gfCNCPoint3[22820] = {X 293.7166, Y 53.8663, Z -4.6667, A 0.000, B 0.000, C 0.000 }
gfCNCPoint3[22821] = {X 294.6128, Y 54.1799, Z -4.6667, A 0.000, B 0.000, C 0.000 }
gfCNCPoint3[22822] = {X 295.4167, Y 54.6850, Z -4.6667, A 0.000, B 0.000, C 0.000 }
gfCNCPoint3[22823] = {X 296.0881, Y 55.3564, Z -4.6667, A 0.000, B 0.000, C 0.000 }
gfCNCPoint3[22824] = {X 296.5932, Y 56.1603, Z -4.6667, A 0.000, B 0.000, C 0.000 }
gfCNCPoint3[22825] = {X 296.9068, Y 57.0565, Z -4.6667, A 0.000, B 0.000, C 0.000 }
gfCNCPoint3[22826] = {X 297.0131, Y 58.0000, Z -4.6667, A 0.000, B 0.000, C 0.000 }
gfCNCPoint3[22827] = {X 297.0131, Y 58.9348, Z -4.6667, A 0.000, B 0.000, C 0.000 }
gfCNCPoint3[22828] = {X 296.9205, Y 59.8045, Z -4.6667, A 0.000, B 0.000, C 0.000 }
gfCNCPoint3[22829] = {X 296.6522, Y 60.6370, Z -4.6667, A 0.000, B 0.000, C 0.000 }
gfCNCPoint3[22830] = {X 296.2193, Y 61.3970, Z -4.6667, A 0.000, B 0.000, C 0.000 }
gfCNCPoint3[22831] = {X 295.6403, Y 62.0524, Z -4.6667, A 0.000, B 0.000, C 0.000 }
gfCNCPoint3[22832] = {X 294.9395, Y 62.5757, Z -4.6667, A 0.000, B 0.000, C 0.000 }
gfCNCPoint3[22833] = {X 294.1465, Y 62.9448, Z -4.6667, A 0.000, B 0.000, C 0.000 }
gfCNCPoint3[22834] = {X 293.2949, Y 63.1439, Z -4.6667, A 0.000, B 0.000, C 0.000 }
gfCNCPoint3[22835] = {X 293.3045, Y 92.8506, Z -4.6667, A 0.000, B 0.000, C 0.000 }
gfCNCPoint3[22836] = {X 294.1540, Y 93.0538, Z -4.6667, A 0.000, B 0.000, C 0.000 }
gfCNCPoint3[22837] = {X 294.9444, Y 93.4255, Z -4.6667, A 0.000, B 0.000, C 0.000 }
gfCNCPoint3[22838] = {X 295.6427, Y 93.9502, Z -4.6667, A 0.000, B 0.000, C 0.000 }
gfCNCPoint3[22839] = {X 296.2197, Y 94.6059, Z -4.6667, A 0.000, B 0.000, C 0.000 }
gfCNCPoint3[22840] = {X 296.6513, Y 95.3652, Z -4.6667, A 0.000, B 0.000, C 0.000 }
gfCNCPoint3[22841] = {X 296.9195, Y 96.1965, Z -4.6667, A 0.000, B 0.000, C 0.000 }
gfCNCPoint3[22842] = {X 297.0131, Y 97.0649, Z -4.6667, A 0.000, B 0.000, C 0.000 }
gfCNCPoint3[22843] = {X 297.0131, Y 98.0000, Z -4.6667, A 0.000, B 0.000, C 0.000 }
gfCNCPoint3[22844] = {X 296.9068, Y 98.9435, Z -4.6667, A 0.000, B 0.000, C 0.000 }
gfCNCPoint3[22845] = {X 296.5932, Y 99.8397, Z -4.6667, A 0.000, B 0.000, C 0.000 }
gfCNCPoint3[22846] = {X 296.0881, Y 100.6436, Z -4.6667, A 0.000, B 0.000, C 0.000 }
gfCNCPoint3[22847] = {X 295.4167, Y 101.3150, Z -4.6667, A 0.000, B 0.000, C 0.000 }
gfCNCPoint3[22848] = {X 294.6128, Y 101.8201, Z -4.6667, A 0.000, B 0.000, C 0.000 }
gfCNCPoint3[22849] = {X 293.7166, Y 102.1337, Z -4.6667, A 0.000, B 0.000, C 0.000 }
gfCNCPoint3[22850] = {X 292.7731, Y 102.2400, Z -4.6667, A 0.000, B 0.000, C 0.000 }
gfCNCPoint3[22851] = {X 276.2327, Y 102.2400, Z -4.6667, A 0.000, B 0.000, C 0.000 }
gfCNCPoint3[22852] = {X 275.2892, Y 102.1337, Z -4.6667, A 0.000, B 0.000, C 0.000 }
gfCNCPoint3[22853] = {X 274.3930, Y 101.8201, Z -4.6667, A 0.000, B 0.000, C 0.000 }
gfCNCPoint3[22854] = {X 273.5891, Y 101.3150, Z -4.6667, A 0.000, B 0.000, C 0.000 }
gfCNCPoint3[22855] = {X 272.9177, Y 100.6436, Z -4.6667, A 0.000, B 0.000, C 0.000 }
gfCNCPoint3[22856] = {X 272.4126, Y 99.8397, Z -4.6667, A 0.000, B 0.000, C 0.000 }
gfCNCPoint3[22857] = {X 272.0990, Y 98.9435, Z -4.6667, A 0.000, B 0.000, C 0.000 }
gfCNCPoint3[22858] = {X 271.9927, Y 98.0000, Z -4.6667, A 0.000, B 0.000, C 0.000 }
gfCNCPoint3[22859] = {X 271.9927, Y 97.0659, Z -4.6667, A 0.000, B 0.000, C 0.000 }
gfCNCPoint3[22860] = {X 272.0830, Y 96.1956, Z -4.6667, A 0.000, B 0.000, C 0.000 }
gfCNCPoint3[22861] = {X 272.3500, Y 95.3624, Z -4.6667, A 0.000, B 0.000, C 0.000 }
gfCNCPoint3[22862] = {X 272.7823, Y 94.6017, Z -4.6667, A 0.000, B 0.000, C 0.000 }
gfCNCPoint3[22863] = {X 273.3615, Y 93.9460, Z -4.6667, A 0.000, B 0.000, C 0.000 }
gfCNCPoint3[22864] = {X 274.0630, Y 93.4231, Z -4.6667, A 0.000, B 0.000, C 0.000 }
gfCNCPoint3[22865] = {X 274.8569, Y 93.0553, Z -4.6667, A 0.000, B 0.000, C 0.000 }
gfCNCPoint3[22866] = {X 275.7094, Y 92.8584, Z -4.6667, A 0.000, B 0.000, C 0.000 }
gfCNCPoint3[22867] = {X 275.7094, Y 85.5404, Z -4.6667, A 0.000, B 0.000, C 0.000 }
gfCNCPoint3[22868] = {X 262.6312, Y 80.4137, Z -4.6667, A 0.000, B 0.000, C 0.000 }
gfCNCPoint3[22869] = {X 262.2340, Y 80.6642, Z -4.6667, A 0.000, B 0.000, C 0.000 }
gfCNCPoint3[22870] = {X 237.7164, Y 96.5448, Z -4.6667, A 0.000, B 0.000, C 0.000 }
gfCNCPoint3[22871] = {X 237.7198, Y 97.0651, Z -4.6667, A 0.000, B 0.000, C 0.000 }
gfCNCPoint3[22872] = {X 237.7198, Y 98.0000, Z -4.6667, A 0.000, B 0.000, C 0.000 }
gfCNCPoint3[22873] = {X 237.6135, Y 98.9435, Z -4.6667, A 0.000, B 0.000, C 0.000 }
gfCNCPoint3[22874] = {X 237.2999, Y 99.8397, Z -4.6667, A 0.000, B 0.000, C 0.000 }
gfCNCPoint3[22875] = {X 236.7948, Y 100.6436, Z -4.6667, A 0.000, B 0.000, C 0.000 }
gfCNCPoint3[22876] = {X 236.1234, Y 101.3150, Z -4.6667, A 0.000, B 0.000, C 0.000 }
gfCNCPoint3[22877] = {X 235.3195, Y 101.8201, Z -4.6667, A 0.000, B 0.000, C 0.000 }
gfCNCPoint3[22878] = {X 234.4233, Y 102.1337, Z -4.6667, A 0.000, B 0.000, C 0.000 }
gfCNCPoint3[22879] = {X 233.4798, Y 102.2400, Z -4.6667, A 0.000, B 0.000, C 0.000 }
gfCNCPoint3[22880] = {X 214.1790, Y 102.2400, Z -4.6667, A 0.000, B 0.000, C 0.000 }
gfCNCPoint3[22881] = {X 213.7861, Y 102.2218, Z -4.6667, A 0.000, B 0.000, C 0.000 }
gfCNCPoint3[22882] = {X 213.3966, Y 102.1672, Z -4.6667, A 0.000, B 0.000, C 0.000 }
gfCNCPoint3[22883] = {X 213.0070, Y 102.2218, Z -4.6667, A 0.000, B 0.000, C 0.000 }
gfCNCPoint3[22884] = {X 212.6141, Y 102.2400, Z -4.6667, A 0.000, B 0.000, C 0.000 }
gfCNCPoint3[22885] = {X 194.9870, Y 102.2400, Z -4.6667, A 0.000, B 0.000, C 0.000 }
gfCNCPoint3[22886] = {X 194.0435, Y 102.1337, Z -4.6667, A 0.000, B 0.000, C 0.000 }
gfCNCPoint3[22887] = {X 193.1473, Y 101.8201, Z -4.6667, A 0.000, B 0.000, C 0.000 }
gfCNCPoint3[22888] = {X 192.3434, Y 101.3150, Z -4.6667, A 0.000, B 0.000, C 0.000 }
gfCNCPoint3[22889] = {X 191.6720, Y 100.6436, Z -4.6667, A 0.000, B 0.000, C 0.000 }
gfCNCPoint3[22890] = {X 191.1669, Y 99.8397, Z -4.6667, A 0.000, B 0.000, C 0.000 }
gfCNCPoint3[22891] = {X 190.8533, Y 98.9435, Z -4.6667, A 0.000, B 0.000, C 0.000 }
gfCNCPoint3[22892] = {X 190.7470, Y 98.0000, Z -4.6667, A 0.000, B 0.000, C 0.000 }
gfCNCPoint3[22893] = {X 190.7470, Y 97.0659, Z -4.6667, A 0.000, B 0.000, C 0.000 }
gfCNCPoint3[22894] = {X 190.8557, Y 96.1118, Z -4.6667, A 0.000, B 0.000, C 0.000 }
gfCNCPoint3[22895] = {X 191.1764, Y 95.2065, Z -4.6667, A 0.000, B 0.000, C 0.000 }
gfCNCPoint3[22896] = {X 191.6926, Y 94.3967, Z -4.6667, A 0.000, B 0.000, C 0.000 }
gfCNCPoint3[22897] = {X 188.5999, Y 91.0202, Z -4.6667, A 0.000, B 0.000, C 0.000 }
gfCNCPoint3[22898] = {X 150.0543, Y 91.0202, Z -4.6667, A 0.000, B 0.000, C 0.000 }
gfCNCPoint3[22899] = {X 147.0396, Y 94.3601, Z -4.6667, A 0.000, B 0.000, C 0.000 }
gfCNCPoint3[22900] = {X 147.5718, Y 95.1783, Z -4.6667, A 0.000, B 0.000, C 0.000 }
gfCNCPoint3[22901] = {X 147.9041, Y 96.0960, Z -4.6667, A 0.000, B 0.000, C 0.000 }
gfCNCPoint3[22902] = {X 148.0191, Y 97.0652, Z -4.6667, A 0.000, B 0.000, C 0.000 }
gfCNCPoint3[22903] = {X 148.0191, Y 98.0000, Z -4.6667, A 0.000, B 0.000, C 0.000 }
gfCNCPoint3[22904] = {X 147.9128, Y 98.9435, Z -4.6667, A 0.000, B 0.000, C 0.000 }
gfCNCPoint3[22905] = {X 147.5992, Y 99.8397, Z -4.6667, A 0.000, B 0.000, C 0.000 }
gfCNCPoint3[22906] = {X 147.0941, Y 100.6436, Z -4.6667, A 0.000, B 0.000, C 0.000 }
gfCNCPoint3[22907] = {X 146.4227, Y 101.3150, Z -4.6667, A 0.000, B 0.000, C 0.000 }
gfCNCPoint3[22908] = {X 145.6188, Y 101.8201, Z -4.6667, A 0.000, B 0.000, C 0.000 }
gfCNCPoint3[22909] = {X 144.7226, Y 102.1337, Z -4.6667, A 0.000, B 0.000, C 0.000 }
gfCNCPoint3[22910] = {X 143.7791, Y 102.2400, Z -4.6667, A 0.000, B 0.000, C 0.000 }
gfCNCPoint3[22911] = {X 125.0000, Y 102.2400, Z -4.6667, A 0.000, B 0.000, C 0.000 }
gfCNCPoint3[22912] = {X 124.0565, Y 102.1337, Z -4.6667, A 0.000, B 0.000, C 0.000 }
gfCNCPoint3[22913] = {X 123.1603, Y 101.8201, Z -4.6667, A 0.000, B 0.000, C 0.000 }
gfCNCPoint3[22914] = {X 122.3564, Y 101.3150, Z -4.6667, A 0.000, B 0.000, C 0.000 }
gfCNCPoint3[22915] = {X 121.6850, Y 100.6436, Z -4.6667, A 0.000, B 0.000, C 0.000 }
gfCNCPoint3[22916] = {X 121.1799, Y 99.8397, Z -4.6667, A 0.000, B 0.000, C 0.000 }
gfCNCPoint3[22917] = {X 120.8663, Y 98.9435, Z -4.6667, A 0.000, B 0.000, C 0.000 }
gfCNCPoint3[22918] = {X 120.7600, Y 98.0000, Z -4.6667, A 0.000, B 0.000, C 0.000 }
gfCNCPoint3[22919] = {X 120.7600, Y 97.0659, Z -4.6667, A 0.000, B 0.000, C 0.000 }
gfCNCPoint3[22920] = {X 120.8618, Y 96.1422, Z -4.6667, A 0.000, B 0.000, C 0.000 }
gfCNCPoint3[22921] = {X 121.1625, Y 95.2629, Z -4.6667, A 0.000, B 0.000, C 0.000 }
gfCNCPoint3[22922] = {X 121.6474, Y 94.4702, Z -4.6667, A 0.000, B 0.000, C 0.000 }
gfCNCPoint3[22923] = {X 122.2934, Y 93.8022, Z -4.6667, A 0.000, B 0.000, C 0.000 }
gfCNCPoint3[22924] = {X 123.0694, Y 93.2910, Z -4.6667, A 0.000, B 0.000, C 0.000 }
gfCNCPoint3[22925] = {X 123.9382, Y 92.9610, Z -4.6667, A 0.000, B 0.000, C 0.000 }
gfCNCPoint3[22926] = {X 124.8579, Y 92.8283, Z -4.6667, A 0.000, B 0.000, C 0.000 }
gfCNCPoint3[22927] = {X 124.8975, Y 92.8108, Z -4.6667, A 0.000, B 0.000, C 0.000 }
gfCNCPoint3[22928] = {X 124.9396, Y 92.8006, Z -4.6667, A 0.000, B 0.000, C 0.000 }
gfCNCPoint3[22929] = {X 125.4606, Y 92.7233, Z -4.6667, A 0.000, B 0.000, C 0.000 }
gfCNCPoint3[22930] = {X 126.3060, Y 92.5807, Z -4.6667, A 0.000, B 0.000, C 0.000 }
gfCNCPoint3[22931] = {X 127.1395, Y 92.3799, Z -4.6667, A 0.000, B 0.000, C 0.000 }
gfCNCPoint3[22932] = {X 128.3715, Y 91.2197, Z -4.6667, A 0.000, B 0.000, C 0.000 }
gfCNCPoint3[22933] = {X 129.5383, Y 89.9938, Z -4.6667, A 0.000, B 0.000, C 0.000 }
gfCNCPoint3[22934] = {X 140.7393, Y 77.6936, Z -4.6667, A 0.000, B 0.000, C 0.000 }
gfCNCPoint3[22935] = {X 137.7818, Y 75.0004, Z -4.6667, A 0.000, B 0.000, C 0.000 }
gfCNCPoint3[22936] = {X 140.7985, Y 77.7475, Z -4.6667, A 0.000, B 0.000, C 0.000 }
gfCNCPoint3[22937] = {X 155.8335, Y 61.2369, Z -4.6667, A 0.000, B 0.000, C 0.000 }
gfCNCPoint3[22938] = {X 155.4565, Y 60.5305, Z -4.6667, A 0.000, B 0.000, C 0.000 }
gfCNCPoint3[22939] = {X 155.2218, Y 59.7648, Z -4.6667, A 0.000, B 0.000, C 0.000 }
gfCNCPoint3[22940] = {X 155.1381, Y 58.9684, Z -4.6667, A 0.000, B 0.000, C 0.000 }
gfCNCPoint3[22941] = {X 155.1380, Y 58.0000, Z -4.6667, A 0.000, B 0.000, C 0.000 }
gfCNCPoint3[22942] = {X 155.2423, Y 57.0743, Z -4.6667, A 0.000, B 0.000, C 0.000 }
gfCNCPoint3[22943] = {X 155.5499, Y 56.1950, Z -4.6667, A 0.000, B 0.000, C 0.000 }
gfCNCPoint3[22944] = {X 156.0455, Y 55.4063, Z -4.6667, A 0.000, B 0.000, C 0.000 }
gfCNCPoint3[22945] = {X 156.7042, Y 54.7476, Z -4.6667, A 0.000, B 0.000, C 0.000 }
gfCNCPoint3[22946] = {X 157.4930, Y 54.2520, Z -4.6667, A 0.000, B 0.000, C 0.000 }
gfCNCPoint3[22947] = {X 158.3723, Y 53.9443, Z -4.6667, A 0.000, B 0.000, C 0.000 }
gfCNCPoint3[22948] = {X 159.2980, Y 53.8400, Z -4.6667, A 0.000, B 0.000, C 0.000 }
gfCNCPoint3[22949] = {X 178.5335, Y 53.8400, Z -4.6667, A 0.000, B 0.000, C 0.000 }
gfCNCPoint3[22950] = {X 179.4592, Y 53.9443, Z -4.6667, A 0.000, B 0.000, C 0.000 }
gfCNCPoint3[22951] = {X 180.3385, Y 54.2520, Z -4.6667, A 0.000, B 0.000, C 0.000 }
gfCNCPoint3[22952] = {X 181.1272, Y 54.7476, Z -4.6667, A 0.000, B 0.000, C 0.000 }
gfCNCPoint3[22953] = {X 181.7859, Y 55.4063, Z -4.6667, A 0.000, B 0.000, C 0.000 }
gfCNCPoint3[22954] = {X 182.2815, Y 56.1950, Z -4.6667, A 0.000, B 0.000, C 0.000 }
gfCNCPoint3[22955] = {X 182.5892, Y 57.0743, Z -4.6667, A 0.000, B 0.000, C 0.000 }
gfCNCPoint3[22956] = {X 182.6935, Y 58.0000, Z -4.6667, A 0.000, B 0.000, C 0.000 }
gfCNCPoint3[22957] = {X 182.6935, Y 58.9342, Z -4.6667, A 0.000, B 0.000, C 0.000 }
gfCNCPoint3[22958] = {X 182.6160, Y 59.7334, Z -4.6667, A 0.000, B 0.000, C 0.000 }
gfCNCPoint3[22959] = {X 182.3864, Y 60.5029, Z -4.6667, A 0.000, B 0.000, C 0.000 }
gfCNCPoint3[22960] = {X 182.0132, Y 61.2138, Z -4.6667, A 0.000, B 0.000, C 0.000 }
gfCNCPoint3[22961] = {X 209.3608, Y 91.0622, Z -4.6667, A 0.000, B 0.000, C 0.000 }
gfCNCPoint3[22962] = {X 210.0261, Y 91.7373, Z -4.6667, A 0.000, B 0.000, C 0.000 }
gfCNCPoint3[22963] = {X 210.7388, Y 92.3620, Z -4.6667, A 0.000, B 0.000, C 0.000 }
gfCNCPoint3[22964] = {X 211.0469, Y 92.5567, Z -4.6667, A 0.000, B 0.000, C 0.000 }
gfCNCPoint3[22965] = {X 211.3924, Y 92.6727, Z -4.6667, A 0.000, B 0.000, C 0.000 }
gfCNCPoint3[22966] = {X 213.3994, Y 92.9858, Z -4.6667, A 0.000, B 0.000, C 0.000 }
gfCNCPoint3[22967] = {X 214.4547, Y 92.8962, Z -4.6667, A 0.000, B 0.000, C 0.000 }
gfCNCPoint3[22968] = {X 215.5121, Y 92.8355, Z -4.6667, A 0.000, B 0.000, C 0.000 }
gfCNCPoint3[22969] = {X 216.2108, Y 92.7589, Z -4.6667, A 0.000, B 0.000, C 0.000 }
gfCNCPoint3[22970] = {X 216.8837, Y 92.5552, Z -4.6667, A 0.000, B 0.000, C 0.000 }
gfCNCPoint3[22971] = {X 217.5077, Y 92.2315, Z -4.6667, A 0.000, B 0.000, C 0.000 }
gfCNCPoint3[22972] = {X 223.0478, Y 88.6562, Z -4.6667, A 0.000, B 0.000, C 0.000 }
gfCNCPoint3[22973] = {X 246.1787, Y 73.8653, Z -4.6667, A 0.000, B 0.000, C 0.000 }
gfCNCPoint3[22974] = {X 221.6899, Y 64.2551, Z -4.6667, A 0.000, B 0.000, C 0.000 }
gfCNCPoint3[22975] = {X 219.9052, Y 63.6577, Z -4.6667, A 0.000, B 0.000, C 0.000 }
gfCNCPoint3[22976] = {X 218.0638, Y 63.2682, Z -4.6667, A 0.000, B 0.000, C 0.000 }
gfCNCPoint3[22977] = {X 216.1900, Y 63.0917, Z -4.6667, A 0.000, B 0.000, C 0.000 }
gfCNCPoint3[22978] = {X 215.2926, Y 62.9624, Z -4.6667, A 0.000, B 0.000, C 0.000 }
gfCNCPoint3[22979] = {X 214.4445, Y 62.6418, Z -4.6667, A 0.000, B 0.000, C 0.000 }
gfCNCPoint3[22980] = {X 213.6860, Y 62.1451, Z -4.6667, A 0.000, B 0.000, C 0.000 }
gfCNCPoint3[22981] = {X 213.0531, Y 61.4958, Z -4.6667, A 0.000, B 0.000, C 0.000 }
gfCNCPoint3[22982] = {X 212.5760, Y 60.7249, Z -4.6667, A 0.000, B 0.000, C 0.000 }
gfCNCPoint3[22983] = {X 212.2772, Y 59.8688, Z -4.6667, A 0.000, B 0.000, C 0.000 }
gfCNCPoint3[22984] = {X 212.1710, Y 58.9684, Z -4.6667, A 0.000, B 0.000, C 0.000 }
gfCNCPoint3[22985] = {X 212.1708, Y 58.0000, Z -4.6667, A 0.000, B 0.000, C 0.000 }
gfCNCPoint3[22986] = {X 212.2751, Y 57.0743, Z -4.6667, A 0.000, B 0.000, C 0.000 }
gfCNCPoint3[22987] = {X 212.5828, Y 56.1950, Z -4.6667, A 0.000, B 0.000, C 0.000 }
gfCNCPoint3[22988] = {X 213.0784, Y 55.4063, Z -4.6667, A 0.000, B 0.000, C 0.000 }
gfCNCPoint3[22989] = {X 213.7371, Y 54.7476, Z -4.6667, A 0.000, B 0.000, C 0.000 }
gfCNCPoint3[22990] = {X 214.5259, Y 54.2520, Z -4.6667, A 0.000, B 0.000, C 0.000 }
gfCNCPoint3[22991] = {X 215.4051, Y 53.9443, Z -4.6667, A 0.000, B 0.000, C 0.000 }
gfCNCPoint3[22992] = {X 216.3308, Y 53.8400, Z -4.6667, A 0.000, B 0.000, C 0.000 }
gfCNCPoint3[22993] = {X 237.2617, Y 53.8400, Z -4.6667, A 0.000, B 0.000, C 0.000 }
gfCNCPoint3[22994] = {X 238.1874, Y 53.9443, Z -4.6667, A 0.000, B 0.000, C 0.000 }
gfCNCPoint3[22995] = {X 239.0666, Y 54.2520, Z -4.6667, A 0.000, B 0.000, C 0.000 }
gfCNCPoint3[22996] = {X 239.8554, Y 54.7476, Z -4.6667, A 0.000, B 0.000, C 0.000 }
gfCNCPoint3[22997] = {X 240.5141, Y 55.4063, Z -4.6667, A 0.000, B 0.000, C 0.000 }
gfCNCPoint3[22998] = {X 241.0097, Y 56.1950, Z -4.6667, A 0.000, B 0.000, C 0.000 }
gfCNCPoint3[22999] = {X 241.3174, Y 57.0743, Z -4.6667, A 0.000, B 0.000, C 0.000 }
gfCNCPoint3[23000] = {X 241.4217, Y 58.0000, Z -4.6667, A 0.000, B 0.000, C 0.000 }
gfCNCPoint3[23001] = {X 241.4217, Y 58.3416, Z -4.6667, A 0.000, B 0.000, C 0.000 }
gfCNCPoint3[23002] = {X 248.0553, Y 60.9282, Z -4.6667, A 0.000, B 0.000, C 0.000 }
gfCNCPoint3[23003] = {X 275.7928, Y 71.9378, Z -4.6667, A 0.000, B 0.000, C 0.000 }
gfCNCPoint3[23004] = {X 275.7940, Y 63.0709, Z -4.6667, A 0.000, B 0.000, C 0.000 }
gfCNCPoint3[23005] = {X 275.6915, Y 63.0587, Z -4.6667, A 0.000, B 0.000, C 0.000 }
gfCNCPoint3[23006] = {X 275.5894, Y 63.0440, Z -4.6667, A 0.000, B 0.000, C 0.000 }
gfCNCPoint3[23007] = {X 274.6519, Y 62.7820, Z -4.6667, A 0.000, B 0.000, C 0.000 }
gfCNCPoint3[23008] = {X 273.8009, Y 62.3093, Z -4.6667, A 0.000, B 0.000, C 0.000 }
gfCNCPoint3[23009] = {X 273.0831, Y 61.6517, Z -4.6667, A 0.000, B 0.000, C 0.000 }
gfCNCPoint3[23010] = {X 272.5377, Y 60.8453, Z -4.6667, A 0.000, B 0.000, C 0.000 }
gfCNCPoint3[23011] = {X 272.1947, Y 59.9342, Z -4.6667, A 0.000, B 0.000, C 0.000 }
gfCNCPoint3[23012] = {X 272.0728, Y 58.9684, Z -4.6667, A 0.000, B 0.000, C 0.000 }
gfCNCPoint3[23013] = {X 272.0727, Y 58.0000, Z -4.6667, A 0.000, B 0.000, C 0.000 }
gfCNCPoint3[23014] = {X 272.1770, Y 57.0743, Z -4.6667, A 0.000, B 0.000, C 0.000 }
gfCNCPoint3[23015] = {X 272.4847, Y 56.1950, Z -4.6667, A 0.000, B 0.000, C 0.000 }
gfCNCPoint3[23016] = {X 272.9803, Y 55.4063, Z -4.6667, A 0.000, B 0.000, C 0.000 }
gfCNCPoint3[23017] = {X 273.6390, Y 54.7476, Z -4.6667, A 0.000, B 0.000, C 0.000 }
gfCNCPoint3[23018] = {X 274.4277, Y 54.2520, Z -4.6667, A 0.000, B 0.000, C 0.000 }
gfCNCPoint3[23019] = {X 275.3070, Y 53.9443, Z -4.6667, A 0.000, B 0.000, C 0.000 }
gfCNCPoint3[23020] = {X 276.2327, Y 53.8400, Z -4.6667, A 0.000, B 0.000, C 0.000 }
gfCNCPoint3[23021] = {X 292.7731, Y 53.8400, Z -4.6667, A 0.000, B 0.000, C 0.000 }
gfCNCPoint3[23022] = {X 293.6988, Y 53.9443, Z -4.6667, A 0.000, B 0.000, C 0.000 }
gfCNCPoint3[23023] = {X 294.5780, Y 54.2520, Z -4.6667, A 0.000, B 0.000, C 0.000 }
gfCNCPoint3[23024] = {X 295.3668, Y 54.7476, Z -4.6667, A 0.000, B 0.000, C 0.000 }
gfCNCPoint3[23025] = {X 296.0255, Y 55.4063, Z -4.6667, A 0.000, B 0.000, C 0.000 }
gfCNCPoint3[23026] = {X 296.5211, Y 56.1950, Z -4.6667, A 0.000, B 0.000, C 0.000 }
gfCNCPoint3[23027] = {X 296.8288, Y 57.0743, Z -4.6667, A 0.000, B 0.000, C 0.000 }
gfCNCPoint3[23028] = {X 296.9331, Y 58.0000, Z -4.6667, A 0.000, B 0.000, C 0.000 }
gfCNCPoint3[23029] = {X 296.9331, Y 58.9346, Z -4.6667, A 0.000, B 0.000, C 0.000 }
gfCNCPoint3[23030] = {X 296.8154, Y 59.9063, Z -4.6667, A 0.000, B 0.000, C 0.000 }
gfCNCPoint3[23031] = {X 296.4747, Y 60.8239, Z -4.6667, A 0.000, B 0.000, C 0.000 }
gfCNCPoint3[23032] = {X 295.9299, Y 61.6370, Z -4.6667, A 0.000, B 0.000, C 0.000 }
gfCNCPoint3[23033] = {X 295.2107, Y 62.3010, Z -4.6667, A 0.000, B 0.000, C 0.000 }
gfCNCPoint3[23034] = {X 294.3568, Y 62.7794, Z -4.6667, A 0.000, B 0.000, C 0.000 }
gfCNCPoint3[23035] = {X 293.4149, Y 63.0459, Z -4.6667, A 0.000, B 0.000, C 0.000 }
gfCNCPoint3[23036] = {X 293.3184, Y 63.0601, Z -4.6667, A 0.000, B 0.000, C 0.000 }
gfCNCPoint3[23037] = {X 293.2216, Y 63.0721, Z -4.6667, A 0.000, B 0.000, C 0.000 }
gfCNCPoint3[23038] = {X 293.2128, Y 63.1618, Z -4.6667, A 0.000, B 0.000, C 0.000 }
gfCNCPoint3[23039] = {X 293.2245, Y 92.9212, Z -4.6667, A 0.000, B 0.000, C 0.000 }
gfCNCPoint3[23040] = {X 293.3195, Y 92.9334, Z -4.6667, A 0.000, B 0.000, C 0.000 }
gfCNCPoint3[23041] = {X 293.4142, Y 92.9477, Z -4.6667, A 0.000, B 0.000, C 0.000 }
gfCNCPoint3[23042] = {X 294.3557, Y 93.2168, Z -4.6667, A 0.000, B 0.000, C 0.000 }
gfCNCPoint3[23043] = {X 295.2090, Y 93.6970, Z -4.6667, A 0.000, B 0.000, C 0.000 }
gfCNCPoint3[23044] = {X 295.9278, Y 94.3620, Z -4.6667, A 0.000, B 0.000, C 0.000 }
gfCNCPoint3[23045] = {X 296.4726, Y 95.1756, Z -4.6667, A 0.000, B 0.000, C 0.000 }
gfCNCPoint3[23046] = {X 296.8140, Y 96.0934, Z -4.6667, A 0.000, B 0.000, C 0.000 }
gfCNCPoint3[23047] = {X 296.9331, Y 97.0653, Z -4.6667, A 0.000, B 0.000, C 0.000 }
gfCNCPoint3[23048] = {X 296.9331, Y 98.0000, Z -4.6667, A 0.000, B 0.000, C 0.000 }
gfCNCPoint3[23049] = {X 296.8288, Y 98.9257, Z -4.6667, A 0.000, B 0.000, C 0.000 }
gfCNCPoint3[23050] = {X 296.5211, Y 99.8050, Z -4.6667, A 0.000, B 0.000, C 0.000 }
gfCNCPoint3[23051] = {X 296.0255, Y 100.5937, Z -4.6667, A 0.000, B 0.000, C 0.000 }
gfCNCPoint3[23052] = {X 295.3668, Y 101.2524, Z -4.6667, A 0.000, B 0.000, C 0.000 }
gfCNCPoint3[23053] = {X 294.5780, Y 101.7480, Z -4.6667, A 0.000, B 0.000, C 0.000 }
gfCNCPoint3[23054] = {X 293.6988, Y 102.0557, Z -4.6667, A 0.000, B 0.000, C 0.000 }
gfCNCPoint3[23055] = {X 292.7731, Y 102.1600, Z -4.6667, A 0.000, B 0.000, C 0.000 }
gfCNCPoint3[23056] = {X 276.2327, Y 102.1600, Z -4.6667, A 0.000, B 0.000, C 0.000 }
gfCNCPoint3[23057] = {X 275.3070, Y 102.0557, Z -4.6667, A 0.000, B 0.000, C 0.000 }
gfCNCPoint3[23058] = {X 274.4277, Y 101.7480, Z -4.6667, A 0.000, B 0.000, C 0.000 }
gfCNCPoint3[23059] = {X 273.6390, Y 101.2524, Z -4.6667, A 0.000, B 0.000, C 0.000 }
gfCNCPoint3[23060] = {X 272.9803, Y 100.5937, Z -4.6667, A 0.000, B 0.000, C 0.000 }
gfCNCPoint3[23061] = {X 272.4847, Y 99.8050, Z -4.6667, A 0.000, B 0.000, C 0.000 }
gfCNCPoint3[23062] = {X 272.1770, Y 98.9257, Z -4.6667, A 0.000, B 0.000, C 0.000 }
gfCNCPoint3[23063] = {X 272.0727, Y 98.0000, Z -4.6667, A 0.000, B 0.000, C 0.000 }
gfCNCPoint3[23064] = {X 272.0727, Y 97.0659, Z -4.6667, A 0.000, B 0.000, C 0.000 }
gfCNCPoint3[23065] = {X 272.1634, Y 96.2022, Z -4.6667, A 0.000, B 0.000, C 0.000 }
gfCNCPoint3[23066] = {X 272.4314, Y 95.3761, Z -4.6667, A 0.000, B 0.000, C 0.000 }
gfCNCPoint3[23067] = {X 272.8651, Y 94.6237, Z -4.6667, A 0.000, B 0.000, C 0.000 }
gfCNCPoint3[23068] = {X 273.4455, Y 93.9777, Z -4.6667, A 0.000, B 0.000, C 0.000 }
gfCNCPoint3[23069] = {X 274.1474, Y 93.4663, Z -4.6667, A 0.000, B 0.000, C 0.000 }
gfCNCPoint3[23070] = {X 274.9403, Y 93.1118, Z -4.6667, A 0.000, B 0.000, C 0.000 }
gfCNCPoint3[23071] = {X 275.7894, Y 92.9296, Z -4.6667, A 0.000, B 0.000, C 0.000 }
gfCNCPoint3[23072] = {X 275.7894, Y 85.4858, Z -4.6667, A 0.000, B 0.000, C 0.000 }
gfCNCPoint3[23073] = {X 262.6228, Y 80.3245, Z -4.6667, A 0.000, B 0.000, C 0.000 }
gfCNCPoint3[23074] = {X 262.1909, Y 80.5968, Z -4.6667, A 0.000, B 0.000, C 0.000 }
gfCNCPoint3[23075] = {X 237.6361, Y 96.5015, Z -4.6667, A 0.000, B 0.000, C 0.000 }
gfCNCPoint3[23076] = {X 237.6398, Y 97.0654, Z -4.6667, A 0.000, B 0.000, C 0.000 }
gfCNCPoint3[23077] = {X 237.6398, Y 98.0000, Z -4.6667, A 0.000, B 0.000, C 0.000 }
gfCNCPoint3[23078] = {X 237.5355, Y 98.9257, Z -4.6667, A 0.000, B 0.000, C 0.000 }
gfCNCPoint3[23079] = {X 237.2278, Y 99.8050, Z -4.6667, A 0.000, B 0.000, C 0.000 }
gfCNCPoint3[23080] = {X 236.7322, Y 100.5937, Z -4.6667, A 0.000, B 0.000, C 0.000 }
gfCNCPoint3[23081] = {X 236.0735, Y 101.2524, Z -4.6667, A 0.000, B 0.000, C 0.000 }
gfCNCPoint3[23082] = {X 235.2847, Y 101.7480, Z -4.6667, A 0.000, B 0.000, C 0.000 }
gfCNCPoint3[23083] = {X 234.4055, Y 102.0557, Z -4.6667, A 0.000, B 0.000, C 0.000 }
gfCNCPoint3[23084] = {X 233.4798, Y 102.1600, Z -4.6667, A 0.000, B 0.000, C 0.000 }
gfCNCPoint3[23085] = {X 214.1790, Y 102.1600, Z -4.6667, A 0.000, B 0.000, C 0.000 }
gfCNCPoint3[23086] = {X 213.7860, Y 102.1414, Z -4.6667, A 0.000, B 0.000, C 0.000 }
gfCNCPoint3[23087] = {X 213.3966, Y 102.0857, Z -4.6667, A 0.000, B 0.000, C 0.000 }
gfCNCPoint3[23088] = {X 213.0071, Y 102.1414, Z -4.6667, A 0.000, B 0.000, C 0.000 }
gfCNCPoint3[23089] = {X 212.6141, Y 102.1600, Z -4.6667, A 0.000, B 0.000, C 0.000 }
gfCNCPoint3[23090] = {X 194.9870, Y 102.1600, Z -4.6667, A 0.000, B 0.000, C 0.000 }
gfCNCPoint3[23091] = {X 194.0613, Y 102.0557, Z -4.6667, A 0.000, B 0.000, C 0.000 }
gfCNCPoint3[23092] = {X 193.1820, Y 101.7480, Z -4.6667, A 0.000, B 0.000, C 0.000 }
gfCNCPoint3[23093] = {X 192.3932, Y 101.2524, Z -4.6667, A 0.000, B 0.000, C 0.000 }
gfCNCPoint3[23094] = {X 191.7345, Y 100.5937, Z -4.6667, A 0.000, B 0.000, C 0.000 }
gfCNCPoint3[23095] = {X 191.2389, Y 99.8050, Z -4.6667, A 0.000, B 0.000, C 0.000 }
gfCNCPoint3[23096] = {X 190.9313, Y 98.9257, Z -4.6667, A 0.000, B 0.000, C 0.000 }
gfCNCPoint3[23097] = {X 190.8270, Y 98.0000, Z -4.6667, A 0.000, B 0.000, C 0.000 }
gfCNCPoint3[23098] = {X 190.8270, Y 97.0659, Z -4.6667, A 0.000, B 0.000, C 0.000 }
gfCNCPoint3[23099] = {X 190.9241, Y 96.1723, Z -4.6667, A 0.000, B 0.000, C 0.000 }
gfCNCPoint3[23100] = {X 191.2109, Y 95.3203, Z -4.6667, A 0.000, B 0.000, C 0.000 }
gfCNCPoint3[23101] = {X 191.6741, Y 94.5499, Z -4.6667, A 0.000, B 0.000, C 0.000 }
gfCNCPoint3[23102] = {X 191.7354, Y 94.4712, Z -4.6667, A 0.000, B 0.000, C 0.000 }
gfCNCPoint3[23103] = {X 191.7986, Y 94.3939, Z -4.6667, A 0.000, B 0.000, C 0.000 }
gfCNCPoint3[23104] = {X 188.6351, Y 90.9402, Z -4.6667, A 0.000, B 0.000, C 0.000 }
gfCNCPoint3[23105] = {X 150.0187, Y 90.9402, Z -4.6667, A 0.000, B 0.000, C 0.000 }
gfCNCPoint3[23106] = {X 146.9335, Y 94.3582, Z -4.6667, A 0.000, B 0.000, C 0.000 }
gfCNCPoint3[23107] = {X 147.4794, Y 95.1728, Z -4.6667, A 0.000, B 0.000, C 0.000 }
gfCNCPoint3[23108] = {X 147.8209, Y 96.0921, Z -4.6667, A 0.000, B 0.000, C 0.000 }
gfCNCPoint3[23109] = {X 147.9391, Y 97.0655, Z -4.6667, A 0.000, B 0.000, C 0.000 }
gfCNCPoint3[23110] = {X 147.9391, Y 98.0000, Z -4.6667, A 0.000, B 0.000, C 0.000 }
gfCNCPoint3[23111] = {X 147.8348, Y 98.9257, Z -4.6667, A 0.000, B 0.000, C 0.000 }
gfCNCPoint3[23112] = {X 147.5271, Y 99.8050, Z -4.6667, A 0.000, B 0.000, C 0.000 }
gfCNCPoint3[23113] = {X 147.0315, Y 100.5937, Z -4.6667, A 0.000, B 0.000, C 0.000 }
gfCNCPoint3[23114] = {X 146.3728, Y 101.2524, Z -4.6667, A 0.000, B 0.000, C 0.000 }
gfCNCPoint3[23115] = {X 145.5841, Y 101.7480, Z -4.6667, A 0.000, B 0.000, C 0.000 }
gfCNCPoint3[23116] = {X 144.7048, Y 102.0557, Z -4.6667, A 0.000, B 0.000, C 0.000 }
gfCNCPoint3[23117] = {X 143.7791, Y 102.1600, Z -4.6667, A 0.000, B 0.000, C 0.000 }
gfCNCPoint3[23118] = {X 125.0000, Y 102.1600, Z -4.6667, A 0.000, B 0.000, C 0.000 }
gfCNCPoint3[23119] = {X 124.0743, Y 102.0557, Z -4.6667, A 0.000, B 0.000, C 0.000 }
gfCNCPoint3[23120] = {X 123.1950, Y 101.7480, Z -4.6667, A 0.000, B 0.000, C 0.000 }
gfCNCPoint3[23121] = {X 122.4063, Y 101.2524, Z -4.6667, A 0.000, B 0.000, C 0.000 }
gfCNCPoint3[23122] = {X 121.7476, Y 100.5937, Z -4.6667, A 0.000, B 0.000, C 0.000 }
gfCNCPoint3[23123] = {X 121.2520, Y 99.8050, Z -4.6667, A 0.000, B 0.000, C 0.000 }
gfCNCPoint3[23124] = {X 120.9443, Y 98.9257, Z -4.6667, A 0.000, B 0.000, C 0.000 }
gfCNCPoint3[23125] = {X 120.8400, Y 98.0000, Z -4.6667, A 0.000, B 0.000, C 0.000 }
gfCNCPoint3[23126] = {X 120.8400, Y 97.0659, Z -4.6667, A 0.000, B 0.000, C 0.000 }
gfCNCPoint3[23127] = {X 120.9406, Y 96.1567, Z -4.6667, A 0.000, B 0.000, C 0.000 }
gfCNCPoint3[23128] = {X 121.2375, Y 95.2914, Z -4.6667, A 0.000, B 0.000, C 0.000 }
gfCNCPoint3[23129] = {X 121.7163, Y 94.5120, Z -4.6667, A 0.000, B 0.000, C 0.000 }
gfCNCPoint3[23130] = {X 122.3539, Y 93.8560, Z -4.6667, A 0.000, B 0.000, C 0.000 }
gfCNCPoint3[23131] = {X 123.1194, Y 93.3553, Z -4.6667, A 0.000, B 0.000, C 0.000 }
gfCNCPoint3[23132] = {X 123.9759, Y 93.0339, Z -4.6667, A 0.000, B 0.000, C 0.000 }
gfCNCPoint3[23133] = {X 124.8820, Y 92.9076, Z -4.6667, A 0.000, B 0.000, C 0.000 }
gfCNCPoint3[23134] = {X 124.9150, Y 92.8896, Z -4.6667, A 0.000, B 0.000, C 0.000 }
gfCNCPoint3[23135] = {X 124.9513, Y 92.8797, Z -4.6667, A 0.000, B 0.000, C 0.000 }
gfCNCPoint3[23136] = {X 125.4717, Y 92.8025, Z -4.6667, A 0.000, B 0.000, C 0.000 }
gfCNCPoint3[23137] = {X 126.3314, Y 92.6572, Z -4.6667, A 0.000, B 0.000, C 0.000 }
gfCNCPoint3[23138] = {X 127.1788, Y 92.4520, Z -4.6667, A 0.000, B 0.000, C 0.000 }
gfCNCPoint3[23139] = {X 128.4214, Y 91.2829, Z -4.6667, A 0.000, B 0.000, C 0.000 }
gfCNCPoint3[23140] = {X 129.5978, Y 90.0473, Z -4.6667, A 0.000, B 0.000, C 0.000 }
gfCNCPoint3[23141] = {X 140.7985, Y 77.7475, Z -4.6667, A 0.000, B 0.000, C 0.000 }
gfCNCPoint3[23142] = {X 137.8410, Y 75.0543, Z -4.6667, A 0.000, B 0.000, C 0.000 }
gfCNCPoint3[23143] = {X 140.8576, Y 77.8013, Z -4.6667, A 0.000, B 0.000, C 0.000 }
gfCNCPoint3[23144] = {X 155.9350, Y 61.2443, Z -4.6667, A 0.000, B 0.000, C 0.000 }
gfCNCPoint3[23145] = {X 155.5465, Y 60.5380, Z -4.6667, A 0.000, B 0.000, C 0.000 }
gfCNCPoint3[23146] = {X 155.3043, Y 59.7692, Z -4.6667, A 0.000, B 0.000, C 0.000 }
gfCNCPoint3[23147] = {X 155.2181, Y 58.9678, Z -4.6667, A 0.000, B 0.000, C 0.000 }
gfCNCPoint3[23148] = {X 155.2180, Y 58.0000, Z -4.6667, A 0.000, B 0.000, C 0.000 }
gfCNCPoint3[23149] = {X 155.3203, Y 57.0921, Z -4.6667, A 0.000, B 0.000, C 0.000 }
gfCNCPoint3[23150] = {X 155.6220, Y 56.2298, Z -4.6667, A 0.000, B 0.000, C 0.000 }
gfCNCPoint3[23151] = {X 156.1081, Y 55.4562, Z -4.6667, A 0.000, B 0.000, C 0.000 }
gfCNCPoint3[23152] = {X 156.7541, Y 54.8101, Z -4.6667, A 0.000, B 0.000, C 0.000 }
gfCNCPoint3[23153] = {X 157.5277, Y 54.3240, Z -4.6667, A 0.000, B 0.000, C 0.000 }
gfCNCPoint3[23154] = {X 158.3901, Y 54.0223, Z -4.6667, A 0.000, B 0.000, C 0.000 }
gfCNCPoint3[23155] = {X 159.2980, Y 53.9200, Z -4.6667, A 0.000, B 0.000, C 0.000 }
gfCNCPoint3[23156] = {X 178.5335, Y 53.9200, Z -4.6667, A 0.000, B 0.000, C 0.000 }
gfCNCPoint3[23157] = {X 179.4414, Y 54.0223, Z -4.6667, A 0.000, B 0.000, C 0.000 }
gfCNCPoint3[23158] = {X 180.3037, Y 54.3240, Z -4.6667, A 0.000, B 0.000, C 0.000 }
gfCNCPoint3[23159] = {X 181.0773, Y 54.8101, Z -4.6667, A 0.000, B 0.000, C 0.000 }
gfCNCPoint3[23160] = {X 181.7234, Y 55.4562, Z -4.6667, A 0.000, B 0.000, C 0.000 }
gfCNCPoint3[23161] = {X 182.2095, Y 56.2298, Z -4.6667, A 0.000, B 0.000, C 0.000 }
gfCNCPoint3[23162] = {X 182.5112, Y 57.0921, Z -4.6667, A 0.000, B 0.000, C 0.000 }
gfCNCPoint3[23163] = {X 182.6135, Y 58.0000, Z -4.6667, A 0.000, B 0.000, C 0.000 }
gfCNCPoint3[23164] = {X 182.6135, Y 58.9342, Z -4.6667, A 0.000, B 0.000, C 0.000 }
gfCNCPoint3[23165] = {X 182.5334, Y 59.7384, Z -4.6667, A 0.000, B 0.000, C 0.000 }
gfCNCPoint3[23166] = {X 182.2965, Y 60.5109, Z -4.6667, A 0.000, B 0.000, C 0.000 }
gfCNCPoint3[23167] = {X 181.9119, Y 61.2217, Z -4.6667, A 0.000, B 0.000, C 0.000 }
gfCNCPoint3[23168] = {X 209.3018, Y 91.1163, Z -4.6667, A 0.000, B 0.000, C 0.000 }
gfCNCPoint3[23169] = {X 209.9712, Y 91.7954, Z -4.6667, A 0.000, B 0.000, C 0.000 }
gfCNCPoint3[23170] = {X 210.6883, Y 92.4241, Z -4.6667, A 0.000, B 0.000, C 0.000 }
gfCNCPoint3[23171] = {X 211.0135, Y 92.6294, Z -4.6667, A 0.000, B 0.000, C 0.000 }
gfCNCPoint3[23172] = {X 211.3782, Y 92.7514, Z -4.6667, A 0.000, B 0.000, C 0.000 }
gfCNCPoint3[23173] = {X 213.3971, Y 93.0664, Z -4.6667, A 0.000, B 0.000, C 0.000 }
gfCNCPoint3[23174] = {X 214.4548, Y 92.9764, Z -4.6667, A 0.000, B 0.000, C 0.000 }
gfCNCPoint3[23175] = {X 215.5145, Y 92.9155, Z -4.6667, A 0.000, B 0.000, C 0.000 }
gfCNCPoint3[23176] = {X 216.2276, Y 92.8371, Z -4.6667, A 0.000, B 0.000, C 0.000 }
gfCNCPoint3[23177] = {X 216.9142, Y 92.6292, Z -4.6667, A 0.000, B 0.000, C 0.000 }
gfCNCPoint3[23178] = {X 217.5510, Y 92.2988, Z -4.6667, A 0.000, B 0.000, C 0.000 }
gfCNCPoint3[23179] = {X 223.0910, Y 88.7235, Z -4.6667, A 0.000, B 0.000, C 0.000 }
gfCNCPoint3[23180] = {X 246.3540, Y 73.8481, Z -4.6667, A 0.000, B 0.000, C 0.000 }
gfCNCPoint3[23181] = {X 221.7196, Y 64.1809, Z -4.6667, A 0.000, B 0.000, C 0.000 }
gfCNCPoint3[23182] = {X 219.9262, Y 63.5805, Z -4.6667, A 0.000, B 0.000, C 0.000 }
gfCNCPoint3[23183] = {X 218.0758, Y 63.1891, Z -4.6667, A 0.000, B 0.000, C 0.000 }
gfCNCPoint3[23184] = {X 216.1929, Y 63.0117, Z -4.6667, A 0.000, B 0.000, C 0.000 }
gfCNCPoint3[23185] = {X 215.3127, Y 62.8850, Z -4.6667, A 0.000, B 0.000, C 0.000 }
gfCNCPoint3[23186] = {X 214.4809, Y 62.5706, Z -4.6667, A 0.000, B 0.000, C 0.000 }
gfCNCPoint3[23187] = {X 213.7369, Y 62.0834, Z -4.6667, A 0.000, B 0.000, C 0.000 }
gfCNCPoint3[23188] = {X 213.1162, Y 61.4466, Z -4.6667, A 0.000, B 0.000, C 0.000 }
gfCNCPoint3[23189] = {X 212.6482, Y 60.6905, Z -4.6667, A 0.000, B 0.000, C 0.000 }
gfCNCPoint3[23190] = {X 212.3552, Y 59.8509, Z -4.6667, A 0.000, B 0.000, C 0.000 }
gfCNCPoint3[23191] = {X 212.2509, Y 58.9678, Z -4.6667, A 0.000, B 0.000, C 0.000 }
gfCNCPoint3[23192] = {X 212.2508, Y 58.0000, Z -4.6667, A 0.000, B 0.000, C 0.000 }
gfCNCPoint3[23193] = {X 212.3531, Y 57.0921, Z -4.6667, A 0.000, B 0.000, C 0.000 }
gfCNCPoint3[23194] = {X 212.6549, Y 56.2298, Z -4.6667, A 0.000, B 0.000, C 0.000 }
gfCNCPoint3[23195] = {X 213.1409, Y 55.4562, Z -4.6667, A 0.000, B 0.000, C 0.000 }
gfCNCPoint3[23196] = {X 213.7870, Y 54.8101, Z -4.6667, A 0.000, B 0.000, C 0.000 }
gfCNCPoint3[23197] = {X 214.5606, Y 54.3240, Z -4.6667, A 0.000, B 0.000, C 0.000 }
gfCNCPoint3[23198] = {X 215.4229, Y 54.0223, Z -4.6667, A 0.000, B 0.000, C 0.000 }
gfCNCPoint3[23199] = {X 216.3308, Y 53.9200, Z -4.6667, A 0.000, B 0.000, C 0.000 }
gfCNCPoint3[23200] = {X 237.2617, Y 53.9200, Z -4.6667, A 0.000, B 0.000, C 0.000 }
gfCNCPoint3[23201] = {X 238.1696, Y 54.0223, Z -4.6667, A 0.000, B 0.000, C 0.000 }
gfCNCPoint3[23202] = {X 239.0319, Y 54.3240, Z -4.6667, A 0.000, B 0.000, C 0.000 }
gfCNCPoint3[23203] = {X 239.8055, Y 54.8101, Z -4.6667, A 0.000, B 0.000, C 0.000 }
gfCNCPoint3[23204] = {X 240.4516, Y 55.4562, Z -4.6667, A 0.000, B 0.000, C 0.000 }
gfCNCPoint3[23205] = {X 240.9376, Y 56.2298, Z -4.6667, A 0.000, B 0.000, C 0.000 }
gfCNCPoint3[23206] = {X 241.2394, Y 57.0921, Z -4.6667, A 0.000, B 0.000, C 0.000 }
gfCNCPoint3[23207] = {X 241.3417, Y 58.0000, Z -4.6667, A 0.000, B 0.000, C 0.000 }
gfCNCPoint3[23208] = {X 241.3417, Y 58.3963, Z -4.6667, A 0.000, B 0.000, C 0.000 }
gfCNCPoint3[23209] = {X 248.0260, Y 61.0026, Z -4.6667, A 0.000, B 0.000, C 0.000 }
gfCNCPoint3[23210] = {X 275.8728, Y 72.0556, Z -4.6667, A 0.000, B 0.000, C 0.000 }
gfCNCPoint3[23211] = {X 275.8740, Y 62.9983, Z -4.6667, A 0.000, B 0.000, C 0.000 }
gfCNCPoint3[23212] = {X 275.7376, Y 62.9839, Z -4.6667, A 0.000, B 0.000, C 0.000 }
gfCNCPoint3[23213] = {X 275.6018, Y 62.9650, Z -4.6667, A 0.000, B 0.000, C 0.000 }
gfCNCPoint3[23214] = {X 274.6823, Y 62.7080, Z -4.6667, A 0.000, B 0.000, C 0.000 }
gfCNCPoint3[23215] = {X 273.8476, Y 62.2443, Z -4.6667, A 0.000, B 0.000, C 0.000 }
gfCNCPoint3[23216] = {X 273.1436, Y 61.5994, Z -4.6667, A 0.000, B 0.000, C 0.000 }
gfCNCPoint3[23217] = {X 272.6088, Y 60.8085, Z -4.6667, A 0.000, B 0.000, C 0.000 }
gfCNCPoint3[23218] = {X 272.2724, Y 59.9150, Z -4.6667, A 0.000, B 0.000, C 0.000 }
gfCNCPoint3[23219] = {X 272.1528, Y 58.9678, Z -4.6667, A 0.000, B 0.000, C 0.000 }
gfCNCPoint3[23220] = {X 272.1527, Y 58.0000, Z -4.6667, A 0.000, B 0.000, C 0.000 }
gfCNCPoint3[23221] = {X 272.2550, Y 57.0921, Z -4.6667, A 0.000, B 0.000, C 0.000 }
gfCNCPoint3[23222] = {X 272.5567, Y 56.2298, Z -4.6667, A 0.000, B 0.000, C 0.000 }
gfCNCPoint3[23223] = {X 273.0428, Y 55.4562, Z -4.6667, A 0.000, B 0.000, C 0.000 }
gfCNCPoint3[23224] = {X 273.6889, Y 54.8101, Z -4.6667, A 0.000, B 0.000, C 0.000 }
gfCNCPoint3[23225] = {X 274.4624, Y 54.3240, Z -4.6667, A 0.000, B 0.000, C 0.000 }
gfCNCPoint3[23226] = {X 275.3248, Y 54.0223, Z -4.6667, A 0.000, B 0.000, C 0.000 }
gfCNCPoint3[23227] = {X 276.2327, Y 53.9200, Z -4.6667, A 0.000, B 0.000, C 0.000 }
gfCNCPoint3[23228] = {X 292.7731, Y 53.9200, Z -4.6667, A 0.000, B 0.000, C 0.000 }
gfCNCPoint3[23229] = {X 293.6810, Y 54.0223, Z -4.6667, A 0.000, B 0.000, C 0.000 }
gfCNCPoint3[23230] = {X 294.5433, Y 54.3240, Z -4.6667, A 0.000, B 0.000, C 0.000 }
gfCNCPoint3[23231] = {X 295.3169, Y 54.8101, Z -4.6667, A 0.000, B 0.000, C 0.000 }
gfCNCPoint3[23232] = {X 295.9630, Y 55.4562, Z -4.6667, A 0.000, B 0.000, C 0.000 }
gfCNCPoint3[23233] = {X 296.4490, Y 56.2298, Z -4.6667, A 0.000, B 0.000, C 0.000 }
gfCNCPoint3[23234] = {X 296.7508, Y 57.0921, Z -4.6667, A 0.000, B 0.000, C 0.000 }
gfCNCPoint3[23235] = {X 296.8531, Y 58.0000, Z -4.6667, A 0.000, B 0.000, C 0.000 }
gfCNCPoint3[23236] = {X 296.8531, Y 58.9343, Z -4.6667, A 0.000, B 0.000, C 0.000 }
gfCNCPoint3[23237] = {X 296.7376, Y 59.8874, Z -4.6667, A 0.000, B 0.000, C 0.000 }
gfCNCPoint3[23238] = {X 296.4035, Y 60.7875, Z -4.6667, A 0.000, B 0.000, C 0.000 }
gfCNCPoint3[23239] = {X 295.8691, Y 61.5850, Z -4.6667, A 0.000, B 0.000, C 0.000 }
gfCNCPoint3[23240] = {X 295.1637, Y 62.2363, Z -4.6667, A 0.000, B 0.000, C 0.000 }
gfCNCPoint3[23241] = {X 294.3261, Y 62.7055, Z -4.6667, A 0.000, B 0.000, C 0.000 }
gfCNCPoint3[23242] = {X 293.4023, Y 62.9669, Z -4.6667, A 0.000, B 0.000, C 0.000 }
gfCNCPoint3[23243] = {X 293.2756, Y 62.9851, Z -4.6667, A 0.000, B 0.000, C 0.000 }
gfCNCPoint3[23244] = {X 293.1483, Y 62.9993, Z -4.6667, A 0.000, B 0.000, C 0.000 }
gfCNCPoint3[23245] = {X 293.1328, Y 63.1580, Z -4.6667, A 0.000, B 0.000, C 0.000 }
gfCNCPoint3[23246] = {X 293.1446, Y 92.9931, Z -4.6667, A 0.000, B 0.000, C 0.000 }
gfCNCPoint3[23247] = {X 293.2732, Y 93.0079, Z -4.6667, A 0.000, B 0.000, C 0.000 }
gfCNCPoint3[23248] = {X 293.4013, Y 93.0267, Z -4.6667, A 0.000, B 0.000, C 0.000 }
gfCNCPoint3[23249] = {X 294.3248, Y 93.2907, Z -4.6667, A 0.000, B 0.000, C 0.000 }
gfCNCPoint3[23250] = {X 295.1619, Y 93.7617, Z -4.6667, A 0.000, B 0.000, C 0.000 }
gfCNCPoint3[23251] = {X 295.8669, Y 94.4140, Z -4.6667, A 0.000, B 0.000, C 0.000 }
gfCNCPoint3[23252] = {X 296.4014, Y 95.2120, Z -4.6667, A 0.000, B 0.000, C 0.000 }
gfCNCPoint3[23253] = {X 296.7362, Y 96.1123, Z -4.6667, A 0.000, B 0.000, C 0.000 }
gfCNCPoint3[23254] = {X 296.8531, Y 97.0657, Z -4.6667, A 0.000, B 0.000, C 0.000 }
gfCNCPoint3[23255] = {X 296.8531, Y 98.0000, Z -4.6667, A 0.000, B 0.000, C 0.000 }
gfCNCPoint3[23256] = {X 296.7508, Y 98.9079, Z -4.6667, A 0.000, B 0.000, C 0.000 }
gfCNCPoint3[23257] = {X 296.4490, Y 99.7702, Z -4.6667, A 0.000, B 0.000, C 0.000 }
gfCNCPoint3[23258] = {X 295.9630, Y 100.5438, Z -4.6667, A 0.000, B 0.000, C 0.000 }
gfCNCPoint3[23259] = {X 295.3169, Y 101.1899, Z -4.6667, A 0.000, B 0.000, C 0.000 }
gfCNCPoint3[23260] = {X 294.5433, Y 101.6760, Z -4.6667, A 0.000, B 0.000, C 0.000 }
gfCNCPoint3[23261] = {X 293.6810, Y 101.9777, Z -4.6667, A 0.000, B 0.000, C 0.000 }
gfCNCPoint3[23262] = {X 292.7731, Y 102.0800, Z -4.6667, A 0.000, B 0.000, C 0.000 }
gfCNCPoint3[23263] = {X 276.2327, Y 102.0800, Z -4.6667, A 0.000, B 0.000, C 0.000 }
gfCNCPoint3[23264] = {X 275.3248, Y 101.9777, Z -4.6667, A 0.000, B 0.000, C 0.000 }
gfCNCPoint3[23265] = {X 274.4624, Y 101.6760, Z -4.6667, A 0.000, B 0.000, C 0.000 }
gfCNCPoint3[23266] = {X 273.6889, Y 101.1899, Z -4.6667, A 0.000, B 0.000, C 0.000 }
gfCNCPoint3[23267] = {X 273.0428, Y 100.5438, Z -4.6667, A 0.000, B 0.000, C 0.000 }
gfCNCPoint3[23268] = {X 272.5567, Y 99.7702, Z -4.6667, A 0.000, B 0.000, C 0.000 }
gfCNCPoint3[23269] = {X 272.2550, Y 98.9079, Z -4.6667, A 0.000, B 0.000, C 0.000 }
gfCNCPoint3[23270] = {X 272.1527, Y 98.0000, Z -4.6667, A 0.000, B 0.000, C 0.000 }
gfCNCPoint3[23271] = {X 272.1527, Y 97.0659, Z -4.6667, A 0.000, B 0.000, C 0.000 }
gfCNCPoint3[23272] = {X 272.2438, Y 96.2087, Z -4.6667, A 0.000, B 0.000, C 0.000 }
gfCNCPoint3[23273] = {X 272.5129, Y 95.3899, Z -4.6667, A 0.000, B 0.000, C 0.000 }
gfCNCPoint3[23274] = {X 272.9480, Y 94.6458, Z -4.6667, A 0.000, B 0.000, C 0.000 }
gfCNCPoint3[23275] = {X 273.5297, Y 94.0097, Z -4.6667, A 0.000, B 0.000, C 0.000 }
gfCNCPoint3[23276] = {X 274.2321, Y 93.5101, Z -4.6667, A 0.000, B 0.000, C 0.000 }
gfCNCPoint3[23277] = {X 275.0238, Y 93.1692, Z -4.6667, A 0.000, B 0.000, C 0.000 }
gfCNCPoint3[23278] = {X 275.8694, Y 93.0021, Z -4.6667, A 0.000, B 0.000, C 0.000 }
gfCNCPoint3[23279] = {X 275.8694, Y 85.4313, Z -4.6667, A 0.000, B 0.000, C 0.000 }
gfCNCPoint3[23280] = {X 262.6143, Y 80.2353, Z -4.6667, A 0.000, B 0.000, C 0.000 }
gfCNCPoint3[23281] = {X 262.1478, Y 80.5294, Z -4.6667, A 0.000, B 0.000, C 0.000 }
gfCNCPoint3[23282] = {X 237.5558, Y 96.4582, Z -4.6667, A 0.000, B 0.000, C 0.000 }
gfCNCPoint3[23283] = {X 237.5598, Y 97.0656, Z -4.6667, A 0.000, B 0.000, C 0.000 }
gfCNCPoint3[23284] = {X 237.5598, Y 98.0000, Z -4.6667, A 0.000, B 0.000, C 0.000 }
gfCNCPoint3[23285] = {X 237.4575, Y 98.9079, Z -4.6667, A 0.000, B 0.000, C 0.000 }
gfCNCPoint3[23286] = {X 237.1557, Y 99.7702, Z -4.6667, A 0.000, B 0.000, C 0.000 }
gfCNCPoint3[23287] = {X 236.6697, Y 100.5438, Z -4.6667, A 0.000, B 0.000, C 0.000 }
gfCNCPoint3[23288] = {X 236.0236, Y 101.1899, Z -4.6667, A 0.000, B 0.000, C 0.000 }
gfCNCPoint3[23289] = {X 235.2500, Y 101.6760, Z -4.6667, A 0.000, B 0.000, C 0.000 }
gfCNCPoint3[23290] = {X 234.3877, Y 101.9777, Z -4.6667, A 0.000, B 0.000, C 0.000 }
gfCNCPoint3[23291] = {X 233.4798, Y 102.0800, Z -4.6667, A 0.000, B 0.000, C 0.000 }
gfCNCPoint3[23292] = {X 214.1790, Y 102.0800, Z -4.6667, A 0.000, B 0.000, C 0.000 }
gfCNCPoint3[23293] = {X 213.7860, Y 102.0610, Z -4.6667, A 0.000, B 0.000, C 0.000 }
gfCNCPoint3[23294] = {X 213.3966, Y 102.0043, Z -4.6667, A 0.000, B 0.000, C 0.000 }
gfCNCPoint3[23295] = {X 213.0072, Y 102.0610, Z -4.6667, A 0.000, B 0.000, C 0.000 }
gfCNCPoint3[23296] = {X 212.6141, Y 102.0800, Z -4.6667, A 0.000, B 0.000, C 0.000 }
gfCNCPoint3[23297] = {X 194.9870, Y 102.0800, Z -4.6667, A 0.000, B 0.000, C 0.000 }
gfCNCPoint3[23298] = {X 194.0791, Y 101.9777, Z -4.6667, A 0.000, B 0.000, C 0.000 }
gfCNCPoint3[23299] = {X 193.2167, Y 101.6760, Z -4.6667, A 0.000, B 0.000, C 0.000 }
gfCNCPoint3[23300] = {X 192.4431, Y 101.1899, Z -4.6667, A 0.000, B 0.000, C 0.000 }
gfCNCPoint3[23301] = {X 191.7971, Y 100.5438, Z -4.6667, A 0.000, B 0.000, C 0.000 }
gfCNCPoint3[23302] = {X 191.3110, Y 99.7702, Z -4.6667, A 0.000, B 0.000, C 0.000 }
gfCNCPoint3[23303] = {X 191.0093, Y 98.9079, Z -4.6667, A 0.000, B 0.000, C 0.000 }
gfCNCPoint3[23304] = {X 190.9070, Y 98.0000, Z -4.6667, A 0.000, B 0.000, C 0.000 }
gfCNCPoint3[23305] = {X 190.9070, Y 97.0659, Z -4.6667, A 0.000, B 0.000, C 0.000 }
gfCNCPoint3[23306] = {X 191.0022, Y 96.1894, Z -4.6667, A 0.000, B 0.000, C 0.000 }
gfCNCPoint3[23307] = {X 191.2835, Y 95.3539, Z -4.6667, A 0.000, B 0.000, C 0.000 }
gfCNCPoint3[23308] = {X 191.7378, Y 94.5983, Z -4.6667, A 0.000, B 0.000, C 0.000 }
gfCNCPoint3[23309] = {X 191.8199, Y 94.4938, Z -4.6667, A 0.000, B 0.000, C 0.000 }
gfCNCPoint3[23310] = {X 191.9053, Y 94.3920, Z -4.6667, A 0.000, B 0.000, C 0.000 }
gfCNCPoint3[23311] = {X 188.6703, Y 90.8602, Z -4.6667, A 0.000, B 0.000, C 0.000 }
gfCNCPoint3[23312] = {X 149.9831, Y 90.8602, Z -4.6667, A 0.000, B 0.000, C 0.000 }
gfCNCPoint3[23313] = {X 146.8266, Y 94.3573, Z -4.6667, A 0.000, B 0.000, C 0.000 }
gfCNCPoint3[23314] = {X 147.3866, Y 95.1677, Z -4.6667, A 0.000, B 0.000, C 0.000 }
gfCNCPoint3[23315] = {X 147.7375, Y 96.0882, Z -4.6667, A 0.000, B 0.000, C 0.000 }
gfCNCPoint3[23316] = {X 147.8591, Y 97.0658, Z -4.6667, A 0.000, B 0.000, C 0.000 }
gfCNCPoint3[23317] = {X 147.8591, Y 98.0000, Z -4.6667, A 0.000, B 0.000, C 0.000 }
gfCNCPoint3[23318] = {X 147.7568, Y 98.9079, Z -4.6667, A 0.000, B 0.000, C 0.000 }
gfCNCPoint3[23319] = {X 147.4551, Y 99.7702, Z -4.6667, A 0.000, B 0.000, C 0.000 }
gfCNCPoint3[23320] = {X 146.9690, Y 100.5438, Z -4.6667, A 0.000, B 0.000, C 0.000 }
gfCNCPoint3[23321] = {X 146.3229, Y 101.1899, Z -4.6667, A 0.000, B 0.000, C 0.000 }
gfCNCPoint3[23322] = {X 145.5494, Y 101.6760, Z -4.6667, A 0.000, B 0.000, C 0.000 }
gfCNCPoint3[23323] = {X 144.6870, Y 101.9777, Z -4.6667, A 0.000, B 0.000, C 0.000 }
gfCNCPoint3[23324] = {X 143.7791, Y 102.0800, Z -4.6667, A 0.000, B 0.000, C 0.000 }
gfCNCPoint3[23325] = {X 125.0000, Y 102.0800, Z -4.6667, A 0.000, B 0.000, C 0.000 }
gfCNCPoint3[23326] = {X 124.0921, Y 101.9777, Z -4.6667, A 0.000, B 0.000, C 0.000 }
gfCNCPoint3[23327] = {X 123.2298, Y 101.6760, Z -4.6667, A 0.000, B 0.000, C 0.000 }
gfCNCPoint3[23328] = {X 122.4562, Y 101.1899, Z -4.6667, A 0.000, B 0.000, C 0.000 }
gfCNCPoint3[23329] = {X 121.8101, Y 100.5438, Z -4.6667, A 0.000, B 0.000, C 0.000 }
gfCNCPoint3[23330] = {X 121.3240, Y 99.7702, Z -4.6667, A 0.000, B 0.000, C 0.000 }
gfCNCPoint3[23331] = {X 121.0223, Y 98.9079, Z -4.6667, A 0.000, B 0.000, C 0.000 }
gfCNCPoint3[23332] = {X 120.9200, Y 98.0000, Z -4.6667, A 0.000, B 0.000, C 0.000 }
gfCNCPoint3[23333] = {X 120.9200, Y 97.0659, Z -4.6667, A 0.000, B 0.000, C 0.000 }
gfCNCPoint3[23334] = {X 121.0194, Y 96.1710, Z -4.6667, A 0.000, B 0.000, C 0.000 }
gfCNCPoint3[23335] = {X 121.3126, Y 95.3196, Z -4.6667, A 0.000, B 0.000, C 0.000 }
gfCNCPoint3[23336] = {X 121.7855, Y 94.5533, Z -4.6667, A 0.000, B 0.000, C 0.000 }
gfCNCPoint3[23337] = {X 122.4149, Y 93.9094, Z -4.6667, A 0.000, B 0.000, C 0.000 }
gfCNCPoint3[23338] = {X 123.1702, Y 93.4192, Z -4.6667, A 0.000, B 0.000, C 0.000 }
gfCNCPoint3[23339] = {X 124.0147, Y 93.1067, Z -4.6667, A 0.000, B 0.000, C 0.000 }
gfCNCPoint3[23340] = {X 124.9071, Y 92.9870, Z -4.6667, A 0.000, B 0.000, C 0.000 }
gfCNCPoint3[23341] = {X 124.9304, Y 92.9715, Z -4.6667, A 0.000, B 0.000, C 0.000 }
gfCNCPoint3[23342] = {X 124.9631, Y 92.9589, Z -4.6667, A 0.000, B 0.000, C 0.000 }
gfCNCPoint3[23343] = {X 125.4829, Y 92.8818, Z -4.6667, A 0.000, B 0.000, C 0.000 }
gfCNCPoint3[23344] = {X 126.3569, Y 92.7336, Z -4.6667, A 0.000, B 0.000, C 0.000 }
gfCNCPoint3[23345] = {X 127.2182, Y 92.5241, Z -4.6667, A 0.000, B 0.000, C 0.000 }
gfCNCPoint3[23346] = {X 128.4712, Y 91.3462, Z -4.6667, A 0.000, B 0.000, C 0.000 }
gfCNCPoint3[23347] = {X 129.6572, Y 90.1009, Z -4.6667, A 0.000, B 0.000, C 0.000 }
gfCNCPoint3[23348] = {X 140.8576, Y 77.8013, Z -4.6667, A 0.000, B 0.000, C 0.000 }
gfCNCPoint3[23349] = {X 137.8975, Y 75.1058, Z -4.6667, A 0.000, B 0.000, C 0.000 }
gfCNCPoint3[23350] = {X 137.8980, Y 75.1053, Z -4.6667, A 0.000, B 0.000, C 0.000 }
gfCNCPoint3[23351] = {X 140.9142, Y 77.8528, Z -4.6667, A 0.000, B 0.000, C 0.000 }
gfCNCPoint3[23352] = {X 156.0372, Y 61.2509, Z -4.6667, A 0.000, B 0.000, C 0.000 }
gfCNCPoint3[23353] = {X 155.6324, Y 60.5352, Z -4.6667, A 0.000, B 0.000, C 0.000 }
gfCNCPoint3[23354] = {X 155.3825, Y 59.7519, Z -4.6667, A 0.000, B 0.000, C 0.000 }
gfCNCPoint3[23355] = {X 155.2980, Y 58.9340, Z -4.6667, A 0.000, B 0.000, C 0.000 }
gfCNCPoint3[23356] = {X 155.2980, Y 58.0000, Z -4.6667, A 0.000, B 0.000, C 0.000 }
gfCNCPoint3[23357] = {X 155.3982, Y 57.1099, Z -4.6667, A 0.000, B 0.000, C 0.000 }
gfCNCPoint3[23358] = {X 155.6941, Y 56.2645, Z -4.6667, A 0.000, B 0.000, C 0.000 }
gfCNCPoint3[23359] = {X 156.1706, Y 55.5060, Z -4.6667, A 0.000, B 0.000, C 0.000 }
gfCNCPoint3[23360] = {X 156.8040, Y 54.8727, Z -4.6667, A 0.000, B 0.000, C 0.000 }
gfCNCPoint3[23361] = {X 157.5624, Y 54.3961, Z -4.6667, A 0.000, B 0.000, C 0.000 }
gfCNCPoint3[23362] = {X 158.4079, Y 54.1003, Z -4.6667, A 0.000, B 0.000, C 0.000 }
gfCNCPoint3[23363] = {X 159.2980, Y 54.0000, Z -4.6667, A 0.000, B 0.000, C 0.000 }
gfCNCPoint3[23364] = {X 178.5335, Y 54.0000, Z -4.6667, A 0.000, B 0.000, C 0.000 }
gfCNCPoint3[23365] = {X 179.4236, Y 54.1003, Z -4.6667, A 0.000, B 0.000, C 0.000 }
gfCNCPoint3[23366] = {X 180.2690, Y 54.3961, Z -4.6667, A 0.000, B 0.000, C 0.000 }
gfCNCPoint3[23367] = {X 181.0275, Y 54.8727, Z -4.6667, A 0.000, B 0.000, C 0.000 }
gfCNCPoint3[23368] = {X 181.6608, Y 55.5060, Z -4.6667, A 0.000, B 0.000, C 0.000 }
gfCNCPoint3[23369] = {X 182.1374, Y 56.2645, Z -4.6667, A 0.000, B 0.000, C 0.000 }
gfCNCPoint3[23370] = {X 182.4332, Y 57.1099, Z -4.6667, A 0.000, B 0.000, C 0.000 }
gfCNCPoint3[23371] = {X 182.5335, Y 58.0000, Z -4.6667, A 0.000, B 0.000, C 0.000 }
gfCNCPoint3[23372] = {X 182.5334, Y 58.9671, Z -4.6667, A 0.000, B 0.000, C 0.000 }
gfCNCPoint3[23373] = {X 182.4463, Y 59.7646, Z -4.6667, A 0.000, B 0.000, C 0.000 }
gfCNCPoint3[23374] = {X 182.2019, Y 60.5288, Z -4.6667, A 0.000, B 0.000, C 0.000 }
gfCNCPoint3[23375] = {X 181.8099, Y 61.2287, Z -4.6667, A 0.000, B 0.000, C 0.000 }
gfCNCPoint3[23376] = {X 209.2429, Y 91.1703, Z -4.6667, A 0.000, B 0.000, C 0.000 }
gfCNCPoint3[23377] = {X 209.9163, Y 91.8536, Z -4.6667, A 0.000, B 0.000, C 0.000 }
gfCNCPoint3[23378] = {X 210.6378, Y 92.4861, Z -4.6667, A 0.000, B 0.000, C 0.000 }
gfCNCPoint3[23379] = {X 210.9792, Y 92.7017, Z -4.6667, A 0.000, B 0.000, C 0.000 }
gfCNCPoint3[23380] = {X 211.3621, Y 92.8298, Z -4.6667, A 0.000, B 0.000, C 0.000 }
gfCNCPoint3[23381] = {X 212.0545, Y 92.9779, Z -4.6667, A 0.000, B 0.000, C 0.000 }
gfCNCPoint3[23382] = {X 213.3961, Y 93.1469, Z -4.6667, A 0.000, B 0.000, C 0.000 }
gfCNCPoint3[23383] = {X 214.4555, Y 93.0565, Z -4.6667, A 0.000, B 0.000, C 0.000 }
gfCNCPoint3[23384] = {X 215.5170, Y 92.9955, Z -4.6667, A 0.000, B 0.000, C 0.000 }
gfCNCPoint3[23385] = {X 216.2444, Y 92.9153, Z -4.6667, A 0.000, B 0.000, C 0.000 }
gfCNCPoint3[23386] = {X 216.9448, Y 92.7031, Z -4.6667, A 0.000, B 0.000, C 0.000 }
gfCNCPoint3[23387] = {X 217.5944, Y 92.3660, Z -4.6667, A 0.000, B 0.000, C 0.000 }
gfCNCPoint3[23388] = {X 223.1343, Y 88.7908, Z -4.6667, A 0.000, B 0.000, C 0.000 }
gfCNCPoint3[23389] = {X 246.5293, Y 73.8310, Z -4.6667, A 0.000, B 0.000, C 0.000 }
gfCNCPoint3[23390] = {X 221.7493, Y 64.1066, Z -4.6667, A 0.000, B 0.000, C 0.000 }
gfCNCPoint3[23391] = {X 219.9472, Y 63.5033, Z -4.6667, A 0.000, B 0.000, C 0.000 }
gfCNCPoint3[23392] = {X 218.0879, Y 63.1100, Z -4.6667, A 0.000, B 0.000, C 0.000 }
gfCNCPoint3[23393] = {X 216.1958, Y 62.9318, Z -4.6667, A 0.000, B 0.000, C 0.000 }
gfCNCPoint3[23394] = {X 215.3283, Y 62.8064, Z -4.6667, A 0.000, B 0.000, C 0.000 }
gfCNCPoint3[23395] = {X 214.5089, Y 62.4950, Z -4.6667, A 0.000, B 0.000, C 0.000 }
gfCNCPoint3[23396] = {X 213.7770, Y 62.0127, Z -4.6667, A 0.000, B 0.000, C 0.000 }
gfCNCPoint3[23397] = {X 213.1677, Y 61.3825, Z -4.6667, A 0.000, B 0.000, C 0.000 }
gfCNCPoint3[23398] = {X 212.7104, Y 60.6348, Z -4.6667, A 0.000, B 0.000, C 0.000 }
gfCNCPoint3[23399] = {X 212.4268, Y 59.8053, Z -4.6667, A 0.000, B 0.000, C 0.000 }
gfCNCPoint3[23400] = {X 212.3308, Y 58.9341, Z -4.6667, A 0.000, B 0.000, C 0.000 }
gfCNCPoint3[23401] = {X 212.3308, Y 58.0000, Z -4.6667, A 0.000, B 0.000, C 0.000 }
gfCNCPoint3[23402] = {X 212.4311, Y 57.1099, Z -4.6667, A 0.000, B 0.000, C 0.000 }
gfCNCPoint3[23403] = {X 212.7269, Y 56.2645, Z -4.6667, A 0.000, B 0.000, C 0.000 }
gfCNCPoint3[23404] = {X 213.2035, Y 55.5060, Z -4.6667, A 0.000, B 0.000, C 0.000 }
gfCNCPoint3[23405] = {X 213.8368, Y 54.8727, Z -4.6667, A 0.000, B 0.000, C 0.000 }
gfCNCPoint3[23406] = {X 214.5953, Y 54.3961, Z -4.6667, A 0.000, B 0.000, C 0.000 }
gfCNCPoint3[23407] = {X 215.4407, Y 54.1003, Z -4.6667, A 0.000, B 0.000, C 0.000 }
gfCNCPoint3[23408] = {X 216.3308, Y 54.0000, Z -4.6667, A 0.000, B 0.000, C 0.000 }
gfCNCPoint3[23409] = {X 237.2617, Y 54.0000, Z -4.6667, A 0.000, B 0.000, C 0.000 }
gfCNCPoint3[23410] = {X 238.1518, Y 54.1003, Z -4.6667, A 0.000, B 0.000, C 0.000 }
gfCNCPoint3[23411] = {X 238.9972, Y 54.3961, Z -4.6667, A 0.000, B 0.000, C 0.000 }
gfCNCPoint3[23412] = {X 239.7556, Y 54.8727, Z -4.6667, A 0.000, B 0.000, C 0.000 }
gfCNCPoint3[23413] = {X 240.3890, Y 55.5060, Z -4.6667, A 0.000, B 0.000, C 0.000 }
gfCNCPoint3[23414] = {X 240.8656, Y 56.2645, Z -4.6667, A 0.000, B 0.000, C 0.000 }
gfCNCPoint3[23415] = {X 241.1614, Y 57.1099, Z -4.6667, A 0.000, B 0.000, C 0.000 }
gfCNCPoint3[23416] = {X 241.2617, Y 58.0000, Z -4.6667, A 0.000, B 0.000, C 0.000 }
gfCNCPoint3[23417] = {X 241.2617, Y 58.4510, Z -4.6667, A 0.000, B 0.000, C 0.000 }
gfCNCPoint3[23418] = {X 247.9967, Y 61.0771, Z -4.6667, A 0.000, B 0.000, C 0.000 }
gfCNCPoint3[23419] = {X 275.9528, Y 72.1734, Z -4.6667, A 0.000, B 0.000, C 0.000 }
gfCNCPoint3[23420] = {X 275.9523, Y 63.0387, Z -4.6667, A 0.000, B 0.000, C 0.000 }
gfCNCPoint3[23421] = {X 275.9573, Y 62.9246, Z -4.6667, A 0.000, B 0.000, C 0.000 }
gfCNCPoint3[23422] = {X 275.7853, Y 62.9090, Z -4.6667, A 0.000, B 0.000, C 0.000 }
gfCNCPoint3[23423] = {X 275.6141, Y 62.8860, Z -4.6667, A 0.000, B 0.000, C 0.000 }
gfCNCPoint3[23424] = {X 274.7076, Y 62.6319, Z -4.6667, A 0.000, B 0.000, C 0.000 }
gfCNCPoint3[23425] = {X 273.8855, Y 62.1730, Z -4.6667, A 0.000, B 0.000, C 0.000 }
gfCNCPoint3[23426] = {X 273.1934, Y 61.5346, Z -4.6667, A 0.000, B 0.000, C 0.000 }
gfCNCPoint3[23427] = {X 272.6698, Y 60.7522, Z -4.6667, A 0.000, B 0.000, C 0.000 }
gfCNCPoint3[23428] = {X 272.3435, Y 59.8690, Z -4.6667, A 0.000, B 0.000, C 0.000 }
gfCNCPoint3[23429] = {X 272.2327, Y 58.9341, Z -4.6667, A 0.000, B 0.000, C 0.000 }
gfCNCPoint3[23430] = {X 272.2327, Y 58.0000, Z -4.6667, A 0.000, B 0.000, C 0.000 }
gfCNCPoint3[23431] = {X 272.3330, Y 57.1099, Z -4.6667, A 0.000, B 0.000, C 0.000 }
gfCNCPoint3[23432] = {X 272.6288, Y 56.2645, Z -4.6667, A 0.000, B 0.000, C 0.000 }
gfCNCPoint3[23433] = {X 273.1054, Y 55.5060, Z -4.6667, A 0.000, B 0.000, C 0.000 }
gfCNCPoint3[23434] = {X 273.7387, Y 54.8727, Z -4.6667, A 0.000, B 0.000, C 0.000 }
gfCNCPoint3[23435] = {X 274.4972, Y 54.3961, Z -4.6667, A 0.000, B 0.000, C 0.000 }
gfCNCPoint3[23436] = {X 275.3426, Y 54.1003, Z -4.6667, A 0.000, B 0.000, C 0.000 }
gfCNCPoint3[23437] = {X 276.2327, Y 54.0000, Z -4.6667, A 0.000, B 0.000, C 0.000 }
gfCNCPoint3[23438] = {X 292.7731, Y 54.0000, Z -4.6667, A 0.000, B 0.000, C 0.000 }
gfCNCPoint3[23439] = {X 293.6632, Y 54.1003, Z -4.6667, A 0.000, B 0.000, C 0.000 }
gfCNCPoint3[23440] = {X 294.5086, Y 54.3961, Z -4.6667, A 0.000, B 0.000, C 0.000 }
gfCNCPoint3[23441] = {X 295.2670, Y 54.8727, Z -4.6667, A 0.000, B 0.000, C 0.000 }
gfCNCPoint3[23442] = {X 295.9004, Y 55.5060, Z -4.6667, A 0.000, B 0.000, C 0.000 }
gfCNCPoint3[23443] = {X 296.3770, Y 56.2645, Z -4.6667, A 0.000, B 0.000, C 0.000 }
gfCNCPoint3[23444] = {X 296.6728, Y 57.1099, Z -4.6667, A 0.000, B 0.000, C 0.000 }
gfCNCPoint3[23445] = {X 296.7731, Y 58.0000, Z -4.6667, A 0.000, B 0.000, C 0.000 }
gfCNCPoint3[23446] = {X 296.7731, Y 58.9341, Z -4.6667, A 0.000, B 0.000, C 0.000 }
gfCNCPoint3[23447] = {X 296.6599, Y 59.8686, Z -4.6667, A 0.000, B 0.000, C 0.000 }
gfCNCPoint3[23448] = {X 296.3323, Y 60.7510, Z -4.6667, A 0.000, B 0.000, C 0.000 }
gfCNCPoint3[23449] = {X 295.8083, Y 61.5330, Z -4.6667, A 0.000, B 0.000, C 0.000 }
gfCNCPoint3[23450] = {X 295.1167, Y 62.1716, Z -4.6667, A 0.000, B 0.000, C 0.000 }
gfCNCPoint3[23451] = {X 294.2955, Y 62.6316, Z -4.6667, A 0.000, B 0.000, C 0.000 }
gfCNCPoint3[23452] = {X 293.3897, Y 62.8879, Z -4.6667, A 0.000, B 0.000, C 0.000 }
gfCNCPoint3[23453] = {X 293.2328, Y 62.9098, Z -4.6667, A 0.000, B 0.000, C 0.000 }
gfCNCPoint3[23454] = {X 293.0752, Y 62.9254, Z -4.6667, A 0.000, B 0.000, C 0.000 }
gfCNCPoint3[23455] = {X 293.0528, Y 63.1540, Z -4.6667, A 0.000, B 0.000, C 0.000 }
gfCNCPoint3[23456] = {X 293.0528, Y 92.9237, Z -4.6667, A 0.000, B 0.000, C 0.000 }
gfCNCPoint3[23457] = {X 293.0752, Y 93.0671, Z -4.6667, A 0.000, B 0.000, C 0.000 }
gfCNCPoint3[23458] = {X 293.2322, Y 93.0833, Z -4.6667, A 0.000, B 0.000, C 0.000 }
gfCNCPoint3[23459] = {X 293.3885, Y 93.1056, Z -4.6667, A 0.000, B 0.000, C 0.000 }
gfCNCPoint3[23460] = {X 294.2940, Y 93.3645, Z -4.6667, A 0.000, B 0.000, C 0.000 }
gfCNCPoint3[23461] = {X 295.1148, Y 93.8263, Z -4.6667, A 0.000, B 0.000, C 0.000 }
gfCNCPoint3[23462] = {X 295.8061, Y 94.4660, Z -4.6667, A 0.000, B 0.000, C 0.000 }
gfCNCPoint3[23463] = {X 296.3302, Y 95.2485, Z -4.6667, A 0.000, B 0.000, C 0.000 }
gfCNCPoint3[23464] = {X 296.6585, Y 96.1312, Z -4.6667, A 0.000, B 0.000, C 0.000 }
gfCNCPoint3[23465] = {X 296.7731, Y 97.0661, Z -4.6667, A 0.000, B 0.000, C 0.000 }
gfCNCPoint3[23466] = {X 296.7731, Y 98.0000, Z -4.6667, A 0.000, B 0.000, C 0.000 }
gfCNCPoint3[23467] = {X 296.6728, Y 98.8901, Z -4.6667, A 0.000, B 0.000, C 0.000 }
gfCNCPoint3[23468] = {X 296.3770, Y 99.7355, Z -4.6667, A 0.000, B 0.000, C 0.000 }
gfCNCPoint3[23469] = {X 295.9004, Y 100.4940, Z -4.6667, A 0.000, B 0.000, C 0.000 }
gfCNCPoint3[23470] = {X 295.2670, Y 101.1273, Z -4.6667, A 0.000, B 0.000, C 0.000 }
gfCNCPoint3[23471] = {X 294.5086, Y 101.6039, Z -4.6667, A 0.000, B 0.000, C 0.000 }
gfCNCPoint3[23472] = {X 293.6632, Y 101.8997, Z -4.6667, A 0.000, B 0.000, C 0.000 }
gfCNCPoint3[23473] = {X 292.7731, Y 102.0000, Z -4.6667, A 0.000, B 0.000, C 0.000 }
gfCNCPoint3[23474] = {X 276.2327, Y 102.0000, Z -4.6667, A 0.000, B 0.000, C 0.000 }
gfCNCPoint3[23475] = {X 275.3426, Y 101.8997, Z -4.6667, A 0.000, B 0.000, C 0.000 }
gfCNCPoint3[23476] = {X 274.4972, Y 101.6039, Z -4.6667, A 0.000, B 0.000, C 0.000 }
gfCNCPoint3[23477] = {X 273.7387, Y 101.1273, Z -4.6667, A 0.000, B 0.000, C 0.000 }
gfCNCPoint3[23478] = {X 273.1054, Y 100.4940, Z -4.6667, A 0.000, B 0.000, C 0.000 }
gfCNCPoint3[23479] = {X 272.6288, Y 99.7355, Z -4.6667, A 0.000, B 0.000, C 0.000 }
gfCNCPoint3[23480] = {X 272.3330, Y 98.8901, Z -4.6667, A 0.000, B 0.000, C 0.000 }
gfCNCPoint3[23481] = {X 272.2327, Y 98.0000, Z -4.6667, A 0.000, B 0.000, C 0.000 }
gfCNCPoint3[23482] = {X 272.2329, Y 97.0232, Z -4.6667, A 0.000, B 0.000, C 0.000 }
gfCNCPoint3[23483] = {X 272.3321, Y 96.1797, Z -4.6667, A 0.000, B 0.000, C 0.000 }
gfCNCPoint3[23484] = {X 272.6072, Y 95.3761, Z -4.6667, A 0.000, B 0.000, C 0.000 }
gfCNCPoint3[23485] = {X 273.0457, Y 94.6486, Z -4.6667, A 0.000, B 0.000, C 0.000 }
gfCNCPoint3[23486] = {X 273.6280, Y 94.0302, Z -4.6667, A 0.000, B 0.000, C 0.000 }
gfCNCPoint3[23487] = {X 274.3277, Y 93.5487, Z -4.6667, A 0.000, B 0.000, C 0.000 }
gfCNCPoint3[23488] = {X 275.1133, Y 93.2258, Z -4.6667, A 0.000, B 0.000, C 0.000 }
gfCNCPoint3[23489] = {X 275.9494, Y 93.0760, Z -4.6667, A 0.000, B 0.000, C 0.000 }
gfCNCPoint3[23490] = {X 275.9494, Y 85.3767, Z -4.6667, A 0.000, B 0.000, C 0.000 }
gfCNCPoint3[23491] = {X 262.6059, Y 80.1460, Z -4.6667, A 0.000, B 0.000, C 0.000 }
gfCNCPoint3[23492] = {X 262.1047, Y 80.4620, Z -4.6667, A 0.000, B 0.000, C 0.000 }
gfCNCPoint3[23493] = {X 237.4755, Y 96.4149, Z -4.6667, A 0.000, B 0.000, C 0.000 }
gfCNCPoint3[23494] = {X 237.4798, Y 97.0659, Z -4.6667, A 0.000, B 0.000, C 0.000 }
gfCNCPoint3[23495] = {X 237.4798, Y 98.0000, Z -4.6667, A 0.000, B 0.000, C 0.000 }
gfCNCPoint3[23496] = {X 237.3795, Y 98.8901, Z -4.6667, A 0.000, B 0.000, C 0.000 }
gfCNCPoint3[23497] = {X 237.0837, Y 99.7355, Z -4.6667, A 0.000, B 0.000, C 0.000 }
gfCNCPoint3[23498] = {X 236.6071, Y 100.4940, Z -4.6667, A 0.000, B 0.000, C 0.000 }
gfCNCPoint3[23499] = {X 235.9737, Y 101.1273, Z -4.6667, A 0.000, B 0.000, C 0.000 }
gfCNCPoint3[23500] = {X 235.2153, Y 101.6039, Z -4.6667, A 0.000, B 0.000, C 0.000 }
gfCNCPoint3[23501] = {X 234.3699, Y 101.8997, Z -4.6667, A 0.000, B 0.000, C 0.000 }
gfCNCPoint3[23502] = {X 233.4798, Y 102.0000, Z -4.6667, A 0.000, B 0.000, C 0.000 }
gfCNCPoint3[23503] = {X 214.1790, Y 102.0000, Z -4.6667, A 0.000, B 0.000, C 0.000 }
gfCNCPoint3[23504] = {X 213.7859, Y 101.9806, Z -4.6667, A 0.000, B 0.000, C 0.000 }
gfCNCPoint3[23505] = {X 213.3966, Y 101.9227, Z -4.6667, A 0.000, B 0.000, C 0.000 }
gfCNCPoint3[23506] = {X 213.0072, Y 101.9806, Z -4.6667, A 0.000, B 0.000, C 0.000 }
gfCNCPoint3[23507] = {X 212.6141, Y 102.0000, Z -4.6667, A 0.000, B 0.000, C 0.000 }
gfCNCPoint3[23508] = {X 194.9870, Y 102.0000, Z -4.6667, A 0.000, B 0.000, C 0.000 }
gfCNCPoint3[23509] = {X 194.0969, Y 101.8997, Z -4.6667, A 0.000, B 0.000, C 0.000 }
gfCNCPoint3[23510] = {X 193.2514, Y 101.6039, Z -4.6667, A 0.000, B 0.000, C 0.000 }
gfCNCPoint3[23511] = {X 192.4930, Y 101.1273, Z -4.6667, A 0.000, B 0.000, C 0.000 }
gfCNCPoint3[23512] = {X 191.8596, Y 100.4940, Z -4.6667, A 0.000, B 0.000, C 0.000 }
gfCNCPoint3[23513] = {X 191.3831, Y 99.7355, Z -4.6667, A 0.000, B 0.000, C 0.000 }
gfCNCPoint3[23514] = {X 191.0872, Y 98.8901, Z -4.6667, A 0.000, B 0.000, C 0.000 }
gfCNCPoint3[23515] = {X 190.9870, Y 98.0000, Z -4.6667, A 0.000, B 0.000, C 0.000 }
gfCNCPoint3[23516] = {X 190.9870, Y 97.0659, Z -4.6667, A 0.000, B 0.000, C 0.000 }
gfCNCPoint3[23517] = {X 191.0804, Y 96.2066, Z -4.6667, A 0.000, B 0.000, C 0.000 }
gfCNCPoint3[23518] = {X 191.3562, Y 95.3874, Z -4.6667, A 0.000, B 0.000, C 0.000 }
gfCNCPoint3[23519] = {X 191.8015, Y 94.6466, Z -4.6667, A 0.000, B 0.000, C 0.000 }
gfCNCPoint3[23520] = {X 191.9055, Y 94.5176, Z -4.6667, A 0.000, B 0.000, C 0.000 }
gfCNCPoint3[23521] = {X 192.0147, Y 94.3930, Z -4.6667, A 0.000, B 0.000, C 0.000 }
gfCNCPoint3[23522] = {X 188.7055, Y 90.7802, Z -4.6667, A 0.000, B 0.000, C 0.000 }
gfCNCPoint3[23523] = {X 149.9476, Y 90.7802, Z -4.6667, A 0.000, B 0.000, C 0.000 }
gfCNCPoint3[23524] = {X 146.7189, Y 94.3572, Z -4.6667, A 0.000, B 0.000, C 0.000 }
gfCNCPoint3[23525] = {X 147.1687, Y 94.9486, Z -4.6667, A 0.000, B 0.000, C 0.000 }
gfCNCPoint3[23526] = {X 147.5022, Y 95.6126, Z -4.6667, A 0.000, B 0.000, C 0.000 }
gfCNCPoint3[23527] = {X 147.7080, Y 96.3265, Z -4.6667, A 0.000, B 0.000, C 0.000 }
gfCNCPoint3[23528] = {X 147.7791, Y 97.0661, Z -4.6667, A 0.000, B 0.000, C 0.000 }
gfCNCPoint3[23529] = {X 147.7791, Y 98.0000, Z -4.6667, A 0.000, B 0.000, C 0.000 }
gfCNCPoint3[23530] = {X 147.6788, Y 98.8901, Z -4.6667, A 0.000, B 0.000, C 0.000 }
gfCNCPoint3[23531] = {X 147.3830, Y 99.7355, Z -4.6667, A 0.000, B 0.000, C 0.000 }
gfCNCPoint3[23532] = {X 146.9064, Y 100.4940, Z -4.6667, A 0.000, B 0.000, C 0.000 }
gfCNCPoint3[23533] = {X 146.2731, Y 101.1273, Z -4.6667, A 0.000, B 0.000, C 0.000 }
gfCNCPoint3[23534] = {X 145.5146, Y 101.6039, Z -4.6667, A 0.000, B 0.000, C 0.000 }
gfCNCPoint3[23535] = {X 144.6692, Y 101.8997, Z -4.6667, A 0.000, B 0.000, C 0.000 }
gfCNCPoint3[23536] = {X 143.7791, Y 102.0000, Z -4.6667, A 0.000, B 0.000, C 0.000 }
gfCNCPoint3[23537] = {X 125.0000, Y 102.0000, Z -4.6667, A 0.000, B 0.000, C 0.000 }
gfCNCPoint3[23538] = {X 124.1099, Y 101.8997, Z -4.6667, A 0.000, B 0.000, C 0.000 }
gfCNCPoint3[23539] = {X 123.2645, Y 101.6039, Z -4.6667, A 0.000, B 0.000, C 0.000 }
gfCNCPoint3[23540] = {X 122.5060, Y 101.1273, Z -4.6667, A 0.000, B 0.000, C 0.000 }
gfCNCPoint3[23541] = {X 121.8727, Y 100.4940, Z -4.6667, A 0.000, B 0.000, C 0.000 }
gfCNCPoint3[23542] = {X 121.3961, Y 99.7355, Z -4.6667, A 0.000, B 0.000, C 0.000 }
gfCNCPoint3[23543] = {X 121.1003, Y 98.8901, Z -4.6667, A 0.000, B 0.000, C 0.000 }
gfCNCPoint3[23544] = {X 121.0000, Y 98.0000, Z -4.6667, A 0.000, B 0.000, C 0.000 }
gfCNCPoint3[23545] = {X 121.0000, Y 97.0659, Z -4.6667, A 0.000, B 0.000, C 0.000 }
gfCNCPoint3[23546] = {X 121.0981, Y 96.1853, Z -4.6667, A 0.000, B 0.000, C 0.000 }
gfCNCPoint3[23547] = {X 121.3877, Y 95.3479, Z -4.6667, A 0.000, B 0.000, C 0.000 }
gfCNCPoint3[23548] = {X 121.8546, Y 94.5948, Z -4.6667, A 0.000, B 0.000, C 0.000 }
gfCNCPoint3[23549] = {X 122.4758, Y 93.9629, Z -4.6667, A 0.000, B 0.000, C 0.000 }
gfCNCPoint3[23550] = {X 123.2209, Y 93.4834, Z -4.6667, A 0.000, B 0.000, C 0.000 }
gfCNCPoint3[23551] = {X 124.0533, Y 93.1796, Z -4.6667, A 0.000, B 0.000, C 0.000 }
gfCNCPoint3[23552] = {X 124.9321, Y 93.0665, Z -4.6667, A 0.000, B 0.000, C 0.000 }
gfCNCPoint3[23553] = {X 124.9748, Y 93.0380, Z -4.6667, A 0.000, B 0.000, C 0.000 }
gfCNCPoint3[23554] = {X 125.4940, Y 92.9610, Z -4.6667, A 0.000, B 0.000, C 0.000 }
gfCNCPoint3[23555] = {X 126.3824, Y 92.8100, Z -4.6667, A 0.000, B 0.000, C 0.000 }
gfCNCPoint3[23556] = {X 127.2576, Y 92.5961, Z -4.6667, A 0.000, B 0.000, C 0.000 }
gfCNCPoint3[23557] = {X 128.5211, Y 91.4094, Z -4.6667, A 0.000, B 0.000, C 0.000 }
gfCNCPoint3[23558] = {X 129.7166, Y 90.1544, Z -4.6667, A 0.000, B 0.000, C 0.000 }
gfCNCPoint3[23559] = {X 133.8038, Y 85.6585, Z -4.6667, A 0.000, B 0.000, C 0.000 }
gfCNCPoint3[23560] = {X 140.9142, Y 77.8528, Z -4.6667, A 0.000, B 0.000, C 0.000 }
gfCNCPoint3[23561] = {X 137.8980, Y 75.1053, Z -4.6667, A 0.000, B 0.000, C 0.000 }
gfCNCPoint3[23562] = {X 137.8980, Y 75.1053, Z -1.6667, A 0.000, B 0.000, C 0.000 }
gfCNCPoint3[23563] = {X 137.8980, Y 75.1053, Z 11.0000, A 0.000, B 0.000, C 0.000 }
gfCNCPoint3[23564] = {X 167.3809, Y 20.2812, Z 11.0000, A 0.000, B 0.000, C 0.000 }
gfCNCPoint3[23565] = {X 167.3809, Y 20.2812, Z -1.6667, A 0.000, B 0.000, C 0.000 }
gfCNCPoint3[23566] = {X 167.3809, Y 20.2812, Z -4.6667, A 0.000, B 0.000, C 0.000 }
gfCNCPoint3[23567] = {X 171.1581, Y 18.7388, Z -4.6667, A 0.000, B 0.000, C 0.000 }
gfCNCPoint3[23568] = {X 169.8405, Y 15.5121, Z -4.6667, A 0.000, B 0.000, C 0.000 }
gfCNCPoint3[23569] = {X 169.5912, Y 14.6607, Z -4.6667, A 0.000, B 0.000, C 0.000 }
gfCNCPoint3[23570] = {X 169.5212, Y 13.7764, Z -4.6667, A 0.000, B 0.000, C 0.000 }
gfCNCPoint3[23571] = {X 169.6332, Y 12.8964, Z -4.6667, A 0.000, B 0.000, C 0.000 }
gfCNCPoint3[23572] = {X 169.9226, Y 12.0578, Z -4.6667, A 0.000, B 0.000, C 0.000 }
gfCNCPoint3[23573] = {X 170.3773, Y 11.2960, Z -4.6667, A 0.000, B 0.000, C 0.000 }
gfCNCPoint3[23574] = {X 170.9779, Y 10.6432, Z -4.6667, A 0.000, B 0.000, C 0.000 }
gfCNCPoint3[23575] = {X 171.6992, Y 10.1268, Z -4.6667, A 0.000, B 0.000, C 0.000 }
gfCNCPoint3[23576] = {X 172.3295, Y 9.7674, Z -4.6667, A 0.000, B 0.000, C 0.000 }
gfCNCPoint3[23577] = {X 173.2114, Y 9.3960, Z -4.6667, A 0.000, B 0.000, C 0.000 }
gfCNCPoint3[23578] = {X 174.1533, Y 9.2278, Z -4.6667, A 0.000, B 0.000, C 0.000 }
gfCNCPoint3[23579] = {X 175.1092, Y 9.2711, Z -4.6667, A 0.000, B 0.000, C 0.000 }
gfCNCPoint3[23580] = {X 176.0321, Y 9.5237, Z -4.6667, A 0.000, B 0.000, C 0.000 }
gfCNCPoint3[23581] = {X 178.2247, Y 8.6000, Z -4.6667, A 0.000, B 0.000, C 0.000 }
gfCNCPoint3[23582] = {X 180.4987, Y 7.9007, Z -4.6667, A 0.000, B 0.000, C 0.000 }
gfCNCPoint3[23583] = {X 182.8314, Y 7.4327, Z -4.6667, A 0.000, B 0.000, C 0.000 }
gfCNCPoint3[23584] = {X 185.1992, Y 7.2009, Z -4.6667, A 0.000, B 0.000, C 0.000 }
gfCNCPoint3[23585] = {X 187.5783, Y 7.2074, Z -4.6667, A 0.000, B 0.000, C 0.000 }
gfCNCPoint3[23586] = {X 189.9448, Y 7.4523, Z -4.6667, A 0.000, B 0.000, C 0.000 }
gfCNCPoint3[23587] = {X 191.7022, Y 7.8136, Z -4.6667, A 0.000, B 0.000, C 0.000 }
gfCNCPoint3[23588] = {X 193.4131, Y 8.3535, Z -4.6667, A 0.000, B 0.000, C 0.000 }
gfCNCPoint3[23589] = {X 195.0595, Y 9.0662, Z -4.6667, A 0.000, B 0.000, C 0.000 }
gfCNCPoint3[23590] = {X 196.6240, Y 9.9444, Z -4.6667, A 0.000, B 0.000, C 0.000 }
gfCNCPoint3[23591] = {X 198.0900, Y 10.9785, Z -4.6667, A 0.000, B 0.000, C 0.000 }
gfCNCPoint3[23592] = {X 199.1501, Y 11.9215, Z -4.6667, A 0.000, B 0.000, C 0.000 }
gfCNCPoint3[23593] = {X 200.1013, Y 12.9742, Z -4.6667, A 0.000, B 0.000, C 0.000 }
gfCNCPoint3[23594] = {X 200.9323, Y 14.1241, Z -4.6667, A 0.000, B 0.000, C 0.000 }
gfCNCPoint3[23595] = {X 201.6333, Y 15.3575, Z -4.6667, A 0.000, B 0.000, C 0.000 }
gfCNCPoint3[23596] = {X 202.1960, Y 16.6600, Z -4.6667, A 0.000, B 0.000, C 0.000 }
gfCNCPoint3[23597] = {X 202.6702, Y 18.3163, Z -4.6667, A 0.000, B 0.000, C 0.000 }
gfCNCPoint3[23598] = {X 202.9517, Y 20.0160, Z -4.6667, A 0.000, B 0.000, C 0.000 }
gfCNCPoint3[23599] = {X 203.0367, Y 21.7368, Z -4.6667, A 0.000, B 0.000, C 0.000 }
gfCNCPoint3[23600] = {X 202.9241, Y 23.4560, Z -4.6667, A 0.000, B 0.000, C 0.000 }
gfCNCPoint3[23601] = {X 202.6154, Y 25.1510, Z -4.6667, A 0.000, B 0.000, C 0.000 }
gfCNCPoint3[23602] = {X 202.1736, Y 26.5972, Z -4.6667, A 0.000, B 0.000, C 0.000 }
gfCNCPoint3[23603] = {X 201.5488, Y 27.9742, Z -4.6667, A 0.000, B 0.000, C 0.000 }
gfCNCPoint3[23604] = {X 200.7516, Y 29.2591, Z -4.6667, A 0.000, B 0.000, C 0.000 }
gfCNCPoint3[23605] = {X 199.7953, Y 30.4303, Z -4.6667, A 0.000, B 0.000, C 0.000 }
gfCNCPoint3[23606] = {X 198.6957, Y 31.4684, Z -4.6667, A 0.000, B 0.000, C 0.000 }
gfCNCPoint3[23607] = {X 199.4971, Y 31.8096, Z -4.6667, A 0.000, B 0.000, C 0.000 }
gfCNCPoint3[23608] = {X 200.2137, Y 32.3046, Z -4.6667, A 0.000, B 0.000, C 0.000 }
gfCNCPoint3[23609] = {X 200.8164, Y 32.9333, Z -4.6667, A 0.000, B 0.000, C 0.000 }
gfCNCPoint3[23610] = {X 201.2808, Y 33.6702, Z -4.6667, A 0.000, B 0.000, C 0.000 }
gfCNCPoint3[23611] = {X 204.3222, Y 39.9530, Z -4.6667, A 0.000, B 0.000, C 0.000 }
gfCNCPoint3[23612] = {X 204.6427, Y 40.8622, Z -4.6667, A 0.000, B 0.000, C 0.000 }
gfCNCPoint3[23613] = {X 204.7537, Y 41.8197, Z -4.6667, A 0.000, B 0.000, C 0.000 }
gfCNCPoint3[23614] = {X 204.6496, Y 42.7781, Z -4.6667, A 0.000, B 0.000, C 0.000 }
gfCNCPoint3[23615] = {X 204.3355, Y 43.6895, Z -4.6667, A 0.000, B 0.000, C 0.000 }
gfCNCPoint3[23616] = {X 203.8272, Y 44.5085, Z -4.6667, A 0.000, B 0.000, C 0.000 }
gfCNCPoint3[23617] = {X 203.1499, Y 45.1945, Z -4.6667, A 0.000, B 0.000, C 0.000 }
gfCNCPoint3[23618] = {X 202.6137, Y 45.6280, Z -4.6667, A 0.000, B 0.000, C 0.000 }
gfCNCPoint3[23619] = {X 201.9091, Y 46.0918, Z -4.6667, A 0.000, B 0.000, C 0.000 }
gfCNCPoint3[23620] = {X 201.1280, Y 46.4103, Z -4.6667, A 0.000, B 0.000, C 0.000 }
gfCNCPoint3[23621] = {X 200.3000, Y 46.5714, Z -4.6667, A 0.000, B 0.000, C 0.000 }
gfCNCPoint3[23622] = {X 199.4565, Y 46.5690, Z -4.6667, A 0.000, B 0.000, C 0.000 }
gfCNCPoint3[23623] = {X 198.6295, Y 46.4031, Z -4.6667, A 0.000, B 0.000, C 0.000 }
gfCNCPoint3[23624] = {X 196.2991, Y 47.6055, Z -4.6667, A 0.000, B 0.000, C 0.000 }
gfCNCPoint3[23625] = {X 193.8687, Y 48.5902, Z -4.6667, A 0.000, B 0.000, C 0.000 }
gfCNCPoint3[23626] = {X 191.3585, Y 49.3487, Z -4.6667, A 0.000, B 0.000, C 0.000 }
gfCNCPoint3[23627] = {X 189.4154, Y 49.7425, Z -4.6667, A 0.000, B 0.000, C 0.000 }
gfCNCPoint3[23628] = {X 187.4453, Y 49.9648, Z -4.6667, A 0.000, B 0.000, C 0.000 }
gfCNCPoint3[23629] = {X 185.4633, Y 50.0139, Z -4.6667, A 0.000, B 0.000, C 0.000 }
gfCNCPoint3[23630] = {X 183.4847, Y 49.8896, Z -4.6667, A 0.000, B 0.000, C 0.000 }
gfCNCPoint3[23631] = {X 181.5244, Y 49.5927, Z -4.6667, A 0.000, B 0.000, C 0.000 }
gfCNCPoint3[23632] = {X 179.6380, Y 49.1211, Z -4.6667, A 0.000, B 0.000, C 0.000 }
gfCNCPoint3[23633] = {X 177.8176, Y 48.4377, Z -4.6667, A 0.000, B 0.000, C 0.000 }
gfCNCPoint3[23634] = {X 176.0869, Y 47.5512, Z -4.6667, A 0.000, B 0.000, C 0.000 }
gfCNCPoint3[23635] = {X 174.4686, Y 46.4733, Z -4.6667, A 0.000, B 0.000, C 0.000 }
gfCNCPoint3[23636] = {X 173.2357, Y 45.4328, Z -4.6667, A 0.000, B 0.000, C 0.000 }
gfCNCPoint3[23637] = {X 172.1386, Y 44.2500, Z -4.6667, A 0.000, B 0.000, C 0.000 }
gfCNCPoint3[23638] = {X 171.1936, Y 42.9425, Z -4.6667, A 0.000, B 0.000, C 0.000 }
gfCNCPoint3[23639] = {X 170.4146, Y 41.5297, Z -4.6667, A 0.000, B 0.000, C 0.000 }
gfCNCPoint3[23640] = {X 169.8133, Y 40.0327, Z -4.6667, A 0.000, B 0.000, C 0.000 }
gfCNCPoint3[23641] = {X 169.3986, Y 38.4736, Z -4.6667, A 0.000, B 0.000, C 0.000 }
gfCNCPoint3[23642] = {X 169.1766, Y 36.8756, Z -4.6667, A 0.000, B 0.000, C 0.000 }
gfCNCPoint3[23643] = {X 169.0927, Y 35.0415, Z -4.6667, A 0.000, B 0.000, C 0.000 }
gfCNCPoint3[23644] = {X 169.2390, Y 33.2113, Z -4.6667, A 0.000, B 0.000, C 0.000 }
gfCNCPoint3[23645] = {X 169.6133, Y 31.4139, Z -4.6667, A 0.000, B 0.000, C 0.000 }
gfCNCPoint3[23646] = {X 170.2096, Y 29.6774, Z -4.6667, A 0.000, B 0.000, C 0.000 }
gfCNCPoint3[23647] = {X 170.8484, Y 28.3704, Z -4.6667, A 0.000, B 0.000, C 0.000 }
gfCNCPoint3[23648] = {X 171.6562, Y 27.1606, Z -4.6667, A 0.000, B 0.000, C 0.000 }
gfCNCPoint3[23649] = {X 172.6185, Y 26.0696, Z -4.6667, A 0.000, B 0.000, C 0.000 }
gfCNCPoint3[23650] = {X 173.7180, Y 25.1170, Z -4.6667, A 0.000, B 0.000, C 0.000 }
gfCNCPoint3[23651] = {X 174.9349, Y 24.3199, Z -4.6667, A 0.000, B 0.000, C 0.000 }
gfCNCPoint3[23652] = {X 174.1523, Y 23.9323, Z -4.6667, A 0.000, B 0.000, C 0.000 }
gfCNCPoint3[23653] = {X 173.4637, Y 23.3951, Z -4.6667, A 0.000, B 0.000, C 0.000 }
gfCNCPoint3[23654] = {X 172.8971, Y 22.7305, Z -4.6667, A 0.000, B 0.000, C 0.000 }
gfCNCPoint3[23655] = {X 172.4758, Y 21.9655, Z -4.6667, A 0.000, B 0.000, C 0.000 }
gfCNCPoint3[23656] = {X 171.1581, Y 18.7388, Z -4.6667, A 0.000, B 0.000, C 0.000 }
gfCNCPoint3[23657] = {X 167.4550, Y 20.2510, Z -4.6667, A 0.000, B 0.000, C 0.000 }
gfCNCPoint3[23658] = {X 171.2322, Y 18.7085, Z -4.6667, A 0.000, B 0.000, C 0.000 }
gfCNCPoint3[23659] = {X 169.9145, Y 15.4818, Z -4.6667, A 0.000, B 0.000, C 0.000 }
gfCNCPoint3[23660] = {X 169.6699, Y 14.6462, Z -4.6667, A 0.000, B 0.000, C 0.000 }
gfCNCPoint3[23661] = {X 169.6011, Y 13.7783, Z -4.6667, A 0.000, B 0.000, C 0.000 }
gfCNCPoint3[23662] = {X 169.7111, Y 12.9146, Z -4.6667, A 0.000, B 0.000, C 0.000 }
gfCNCPoint3[23663] = {X 169.9952, Y 12.0915, Z -4.6667, A 0.000, B 0.000, C 0.000 }
gfCNCPoint3[23664] = {X 170.4414, Y 11.3439, Z -4.6667, A 0.000, B 0.000, C 0.000 }
gfCNCPoint3[23665] = {X 171.0309, Y 10.7031, Z -4.6667, A 0.000, B 0.000, C 0.000 }
gfCNCPoint3[23666] = {X 171.7389, Y 10.1963, Z -4.6667, A 0.000, B 0.000, C 0.000 }
gfCNCPoint3[23667] = {X 172.3689, Y 9.8371, Z -4.6667, A 0.000, B 0.000, C 0.000 }
gfCNCPoint3[23668] = {X 173.2427, Y 9.4702, Z -4.6667, A 0.000, B 0.000, C 0.000 }
gfCNCPoint3[23669] = {X 174.1762, Y 9.3065, Z -4.6667, A 0.000, B 0.000, C 0.000 }
gfCNCPoint3[23670] = {X 175.1228, Y 9.3543, Z -4.6667, A 0.000, B 0.000, C 0.000 }
gfCNCPoint3[23671] = {X 176.0351, Y 9.6111, Z -4.6667, A 0.000, B 0.000, C 0.000 }
gfCNCPoint3[23672] = {X 178.2244, Y 8.6853, Z -4.6667, A 0.000, B 0.000, C 0.000 }
gfCNCPoint3[23673] = {X 180.4956, Y 7.9840, Z -4.6667, A 0.000, B 0.000, C 0.000 }
gfCNCPoint3[23674] = {X 182.8258, Y 7.5145, Z -4.6667, A 0.000, B 0.000, C 0.000 }
gfCNCPoint3[23675] = {X 185.1913, Y 7.2813, Z -4.6667, A 0.000, B 0.000, C 0.000 }
gfCNCPoint3[23676] = {X 187.5683, Y 7.2870, Z -4.6667, A 0.000, B 0.000, C 0.000 }
gfCNCPoint3[23677] = {X 189.9327, Y 7.5314, Z -4.6667, A 0.000, B 0.000, C 0.000 }
gfCNCPoint3[23678] = {X 191.6820, Y 7.8910, Z -4.6667, A 0.000, B 0.000, C 0.000 }
gfCNCPoint3[23679] = {X 193.3851, Y 8.4284, Z -4.6667, A 0.000, B 0.000, C 0.000 }
gfCNCPoint3[23680] = {X 195.0240, Y 9.1379, Z -4.6667, A 0.000, B 0.000, C 0.000 }
gfCNCPoint3[23681] = {X 196.5813, Y 10.0120, Z -4.6667, A 0.000, B 0.000, C 0.000 }
gfCNCPoint3[23682] = {X 198.0406, Y 11.0415, Z -4.6667, A 0.000, B 0.000, C 0.000 }
gfCNCPoint3[23683] = {X 199.0940, Y 11.9786, Z -4.6667, A 0.000, B 0.000, C 0.000 }
gfCNCPoint3[23684] = {X 200.0393, Y 13.0248, Z -4.6667, A 0.000, B 0.000, C 0.000 }
gfCNCPoint3[23685] = {X 200.8651, Y 14.1675, Z -4.6667, A 0.000, B 0.000, C 0.000 }
gfCNCPoint3[23686] = {X 201.5618, Y 15.3933, Z -4.6667, A 0.000, B 0.000, C 0.000 }
gfCNCPoint3[23687] = {X 202.1210, Y 16.6876, Z -4.6667, A 0.000, B 0.000, C 0.000 }
gfCNCPoint3[23688] = {X 202.5925, Y 18.3350, Z -4.6667, A 0.000, B 0.000, C 0.000 }
gfCNCPoint3[23689] = {X 202.8723, Y 20.0255, Z -4.6667, A 0.000, B 0.000, C 0.000 }
gfCNCPoint3[23690] = {X 202.9567, Y 21.7369, Z -4.6667, A 0.000, B 0.000, C 0.000 }
gfCNCPoint3[23691] = {X 202.8447, Y 23.4467, Z -4.6667, A 0.000, B 0.000, C 0.000 }
gfCNCPoint3[23692] = {X 202.5376, Y 25.1324, Z -4.6667, A 0.000, B 0.000, C 0.000 }
gfCNCPoint3[23693] = {X 202.0881, Y 26.5970, Z -4.6667, A 0.000, B 0.000, C 0.000 }
gfCNCPoint3[23694] = {X 201.4497, Y 27.9897, Z -4.6667, A 0.000, B 0.000, C 0.000 }
gfCNCPoint3[23695] = {X 200.6335, Y 29.2862, Z -4.6667, A 0.000, B 0.000, C 0.000 }
gfCNCPoint3[23696] = {X 199.6538, Y 30.4640, Z -4.6667, A 0.000, B 0.000, C 0.000 }
gfCNCPoint3[23697] = {X 198.5275, Y 31.5026, Z -4.6667, A 0.000, B 0.000, C 0.000 }
gfCNCPoint3[23698] = {X 199.3589, Y 31.8265, Z -4.6667, A 0.000, B 0.000, C 0.000 }
gfCNCPoint3[23699] = {X 200.1041, Y 32.3173, Z -4.6667, A 0.000, B 0.000, C 0.000 }
gfCNCPoint3[23700] = {X 200.7301, Y 32.9531, Z -4.6667, A 0.000, B 0.000, C 0.000 }
gfCNCPoint3[23701] = {X 201.2091, Y 33.7058, Z -4.6667, A 0.000, B 0.000, C 0.000 }
gfCNCPoint3[23702] = {X 204.2502, Y 39.9879, Z -4.6667, A 0.000, B 0.000, C 0.000 }
gfCNCPoint3[23703] = {X 204.5648, Y 40.8802, Z -4.6667, A 0.000, B 0.000, C 0.000 }
gfCNCPoint3[23704] = {X 204.6737, Y 41.8200, Z -4.6667, A 0.000, B 0.000, C 0.000 }
gfCNCPoint3[23705] = {X 204.5715, Y 42.7606, Z -4.6667, A 0.000, B 0.000, C 0.000 }
gfCNCPoint3[23706] = {X 204.2633, Y 43.6551, Z -4.6667, A 0.000, B 0.000, C 0.000 }
gfCNCPoint3[23707] = {X 203.7643, Y 44.4590, Z -4.6667, A 0.000, B 0.000, C 0.000 }
gfCNCPoint3[23708] = {X 203.0996, Y 45.1323, Z -4.6667, A 0.000, B 0.000, C 0.000 }
gfCNCPoint3[23709] = {X 202.5634, Y 45.5658, Z -4.6667, A 0.000, B 0.000, C 0.000 }
gfCNCPoint3[23710] = {X 201.8657, Y 46.0242, Z -4.6667, A 0.000, B 0.000, C 0.000 }
gfCNCPoint3[23711] = {X 201.0919, Y 46.3375, Z -4.6667, A 0.000, B 0.000, C 0.000 }
gfCNCPoint3[23712] = {X 200.2718, Y 46.4936, Z -4.6667, A 0.000, B 0.000, C 0.000 }
gfCNCPoint3[23713] = {X 199.4371, Y 46.4865, Z -4.6667, A 0.000, B 0.000, C 0.000 }
gfCNCPoint3[23714] = {X 198.6198, Y 46.3164, Z -4.6667, A 0.000, B 0.000, C 0.000 }
gfCNCPoint3[23715] = {X 196.8803, Y 47.2416, Z -4.6667, A 0.000, B 0.000, C 0.000 }
gfCNCPoint3[23716] = {X 195.0812, Y 48.0449, Z -4.6667, A 0.000, B 0.000, C 0.000 }
gfCNCPoint3[23717] = {X 193.2312, Y 48.7225, Z -4.6667, A 0.000, B 0.000, C 0.000 }
gfCNCPoint3[23718] = {X 191.3389, Y 49.2712, Z -4.6667, A 0.000, B 0.000, C 0.000 }
gfCNCPoint3[23719] = {X 189.4026, Y 49.6635, Z -4.6667, A 0.000, B 0.000, C 0.000 }
gfCNCPoint3[23720] = {X 187.4395, Y 49.8850, Z -4.6667, A 0.000, B 0.000, C 0.000 }
gfCNCPoint3[23721] = {X 185.4646, Y 49.9339, Z -4.6667, A 0.000, B 0.000, C 0.000 }
gfCNCPoint3[23722] = {X 183.4929, Y 49.8100, Z -4.6667, A 0.000, B 0.000, C 0.000 }
gfCNCPoint3[23723] = {X 181.5396, Y 49.5142, Z -4.6667, A 0.000, B 0.000, C 0.000 }
gfCNCPoint3[23724] = {X 179.6619, Y 49.0448, Z -4.6667, A 0.000, B 0.000, C 0.000 }
gfCNCPoint3[23725] = {X 177.8500, Y 48.3645, Z -4.6667, A 0.000, B 0.000, C 0.000 }
gfCNCPoint3[23726] = {X 176.1274, Y 47.4822, Z -4.6667, A 0.000, B 0.000, C 0.000 }
gfCNCPoint3[23727] = {X 174.5165, Y 46.4093, Z -4.6667, A 0.000, B 0.000, C 0.000 }
gfCNCPoint3[23728] = {X 173.2909, Y 45.3749, Z -4.6667, A 0.000, B 0.000, C 0.000 }
gfCNCPoint3[23729] = {X 172.2003, Y 44.1991, Z -4.6667, A 0.000, B 0.000, C 0.000 }
gfCNCPoint3[23730] = {X 171.2609, Y 42.8993, Z -4.6667, A 0.000, B 0.000, C 0.000 }
gfCNCPoint3[23731] = {X 170.4866, Y 41.4948, Z -4.6667, A 0.000, B 0.000, C 0.000 }
gfCNCPoint3[23732] = {X 169.8889, Y 40.0066, Z -4.6667, A 0.000, B 0.000, C 0.000 }
gfCNCPoint3[23733] = {X 169.4768, Y 38.4567, Z -4.6667, A 0.000, B 0.000, C 0.000 }
gfCNCPoint3[23734] = {X 169.2563, Y 36.8682, Z -4.6667, A 0.000, B 0.000, C 0.000 }
gfCNCPoint3[23735] = {X 169.1726, Y 35.0438, Z -4.6667, A 0.000, B 0.000, C 0.000 }
gfCNCPoint3[23736] = {X 169.3181, Y 33.2232, Z -4.6667, A 0.000, B 0.000, C 0.000 }
gfCNCPoint3[23737] = {X 169.6904, Y 31.4352, Z -4.6667, A 0.000, B 0.000, C 0.000 }
gfCNCPoint3[23738] = {X 170.2836, Y 29.7078, Z -4.6667, A 0.000, B 0.000, C 0.000 }
gfCNCPoint3[23739] = {X 170.9355, Y 28.3796, Z -4.6667, A 0.000, B 0.000, C 0.000 }
gfCNCPoint3[23740] = {X 171.7631, Y 27.1532, Z -4.6667, A 0.000, B 0.000, C 0.000 }
gfCNCPoint3[23741] = {X 172.7510, Y 26.0517, Z -4.6667, A 0.000, B 0.000, C 0.000 }
gfCNCPoint3[23742] = {X 173.8803, Y 25.0958, Z -4.6667, A 0.000, B 0.000, C 0.000 }
gfCNCPoint3[23743] = {X 175.1299, Y 24.3036, Z -4.6667, A 0.000, B 0.000, C 0.000 }
gfCNCPoint3[23744] = {X 174.3084, Y 23.9334, Z -4.6667, A 0.000, B 0.000, C 0.000 }
gfCNCPoint3[23745] = {X 173.5837, Y 23.3981, Z -4.6667, A 0.000, B 0.000, C 0.000 }
gfCNCPoint3[23746] = {X 172.9885, Y 22.7216, Z -4.6667, A 0.000, B 0.000, C 0.000 }
gfCNCPoint3[23747] = {X 172.5496, Y 21.9347, Z -4.6667, A 0.000, B 0.000, C 0.000 }
gfCNCPoint3[23748] = {X 171.2322, Y 18.7085, Z -4.6667, A 0.000, B 0.000, C 0.000 }
gfCNCPoint3[23749] = {X 167.5291, Y 20.2207, Z -4.6667, A 0.000, B 0.000, C 0.000 }
gfCNCPoint3[23750] = {X 171.3062, Y 18.6783, Z -4.6667, A 0.000, B 0.000, C 0.000 }
gfCNCPoint3[23751] = {X 169.9886, Y 15.4516, Z -4.6667, A 0.000, B 0.000, C 0.000 }
gfCNCPoint3[23752] = {X 169.7252, Y 14.4911, Z -4.6667, A 0.000, B 0.000, C 0.000 }
gfCNCPoint3[23753] = {X 169.6977, Y 13.4955, Z -4.6667, A 0.000, B 0.000, C 0.000 }
gfCNCPoint3[23754] = {X 169.9076, Y 12.5218, Z -4.6667, A 0.000, B 0.000, C 0.000 }
gfCNCPoint3[23755] = {X 170.3429, Y 11.6260, Z -4.6667, A 0.000, B 0.000, C 0.000 }
gfCNCPoint3[23756] = {X 170.9787, Y 10.8594, Z -4.6667, A 0.000, B 0.000, C 0.000 }
gfCNCPoint3[23757] = {X 171.7785, Y 10.2658, Z -4.6667, A 0.000, B 0.000, C 0.000 }
gfCNCPoint3[23758] = {X 172.4082, Y 9.9068, Z -4.6667, A 0.000, B 0.000, C 0.000 }
gfCNCPoint3[23759] = {X 173.2740, Y 9.5444, Z -4.6667, A 0.000, B 0.000, C 0.000 }
gfCNCPoint3[23760] = {X 174.1990, Y 9.3853, Z -4.6667, A 0.000, B 0.000, C 0.000 }
gfCNCPoint3[23761] = {X 175.1362, Y 9.4376, Z -4.6667, A 0.000, B 0.000, C 0.000 }
gfCNCPoint3[23762] = {X 176.0377, Y 9.6988, Z -4.6667, A 0.000, B 0.000, C 0.000 }
gfCNCPoint3[23763] = {X 178.2238, Y 8.7707, Z -4.6667, A 0.000, B 0.000, C 0.000 }
gfCNCPoint3[23764] = {X 180.4922, Y 8.0674, Z -4.6667, A 0.000, B 0.000, C 0.000 }
gfCNCPoint3[23765] = {X 182.8199, Y 7.5962, Z -4.6667, A 0.000, B 0.000, C 0.000 }
gfCNCPoint3[23766] = {X 185.1833, Y 7.3618, Z -4.6667, A 0.000, B 0.000, C 0.000 }
gfCNCPoint3[23767] = {X 187.5582, Y 7.3666, Z -4.6667, A 0.000, B 0.000, C 0.000 }
gfCNCPoint3[23768] = {X 189.9205, Y 7.6105, Z -4.6667, A 0.000, B 0.000, C 0.000 }
gfCNCPoint3[23769] = {X 191.6618, Y 7.9684, Z -4.6667, A 0.000, B 0.000, C 0.000 }
gfCNCPoint3[23770] = {X 193.3571, Y 8.5033, Z -4.6667, A 0.000, B 0.000, C 0.000 }
gfCNCPoint3[23771] = {X 194.9884, Y 9.2096, Z -4.6667, A 0.000, B 0.000, C 0.000 }
gfCNCPoint3[23772] = {X 196.5386, Y 10.0797, Z -4.6667, A 0.000, B 0.000, C 0.000 }
gfCNCPoint3[23773] = {X 197.9912, Y 11.1044, Z -4.6667, A 0.000, B 0.000, C 0.000 }
gfCNCPoint3[23774] = {X 199.2832, Y 12.2858, Z -4.6667, A 0.000, B 0.000, C 0.000 }
gfCNCPoint3[23775] = {X 200.4029, Y 13.6317, Z -4.6667, A 0.000, B 0.000, C 0.000 }
gfCNCPoint3[23776] = {X 201.3294, Y 15.1171, Z -4.6667, A 0.000, B 0.000, C 0.000 }
gfCNCPoint3[23777] = {X 202.0457, Y 16.7147, Z -4.6667, A 0.000, B 0.000, C 0.000 }
gfCNCPoint3[23778] = {X 202.5145, Y 18.3531, Z -4.6667, A 0.000, B 0.000, C 0.000 }
gfCNCPoint3[23779] = {X 202.7928, Y 20.0345, Z -4.6667, A 0.000, B 0.000, C 0.000 }
gfCNCPoint3[23780] = {X 202.8767, Y 21.7366, Z -4.6667, A 0.000, B 0.000, C 0.000 }
gfCNCPoint3[23781] = {X 202.7652, Y 23.4372, Z -4.6667, A 0.000, B 0.000, C 0.000 }
gfCNCPoint3[23782] = {X 202.4598, Y 25.1138, Z -4.6667, A 0.000, B 0.000, C 0.000 }
gfCNCPoint3[23783] = {X 202.0019, Y 26.5984, Z -4.6667, A 0.000, B 0.000, C 0.000 }
gfCNCPoint3[23784] = {X 201.3486, Y 28.0081, Z -4.6667, A 0.000, B 0.000, C 0.000 }
gfCNCPoint3[23785] = {X 200.5117, Y 29.3171, Z -4.6667, A 0.000, B 0.000, C 0.000 }
gfCNCPoint3[23786] = {X 199.5065, Y 30.5018, Z -4.6667, A 0.000, B 0.000, C 0.000 }
gfCNCPoint3[23787] = {X 198.3512, Y 31.5407, Z -4.6667, A 0.000, B 0.000, C 0.000 }
gfCNCPoint3[23788] = {X 199.2147, Y 31.8440, Z -4.6667, A 0.000, B 0.000, C 0.000 }
gfCNCPoint3[23789] = {X 199.9909, Y 32.3288, Z -4.6667, A 0.000, B 0.000, C 0.000 }
gfCNCPoint3[23790] = {X 200.6424, Y 32.9717, Z -4.6667, A 0.000, B 0.000, C 0.000 }
gfCNCPoint3[23791] = {X 201.1375, Y 33.7414, Z -4.6667, A 0.000, B 0.000, C 0.000 }
gfCNCPoint3[23792] = {X 204.1781, Y 40.0227, Z -4.6667, A 0.000, B 0.000, C 0.000 }
gfCNCPoint3[23793] = {X 204.4868, Y 40.8982, Z -4.6667, A 0.000, B 0.000, C 0.000 }
gfCNCPoint3[23794] = {X 204.5937, Y 41.8203, Z -4.6667, A 0.000, B 0.000, C 0.000 }
gfCNCPoint3[23795] = {X 204.4934, Y 42.7431, Z -4.6667, A 0.000, B 0.000, C 0.000 }
gfCNCPoint3[23796] = {X 204.1910, Y 43.6208, Z -4.6667, A 0.000, B 0.000, C 0.000 }
gfCNCPoint3[23797] = {X 203.7015, Y 44.4095, Z -4.6667, A 0.000, B 0.000, C 0.000 }
gfCNCPoint3[23798] = {X 203.0493, Y 45.0700, Z -4.6667, A 0.000, B 0.000, C 0.000 }
gfCNCPoint3[23799] = {X 202.5131, Y 45.5036, Z -4.6667, A 0.000, B 0.000, C 0.000 }
gfCNCPoint3[23800] = {X 201.8224, Y 45.9566, Z -4.6667, A 0.000, B 0.000, C 0.000 }
gfCNCPoint3[23801] = {X 201.0559, Y 46.2647, Z -4.6667, A 0.000, B 0.000, C 0.000 }
gfCNCPoint3[23802] = {X 200.2438, Y 46.4158, Z -4.6667, A 0.000, B 0.000, C 0.000 }
gfCNCPoint3[23803] = {X 199.4178, Y 46.4039, Z -4.6667, A 0.000, B 0.000, C 0.000 }
gfCNCPoint3[23804] = {X 198.6103, Y 46.2295, Z -4.6667, A 0.000, B 0.000, C 0.000 }
gfCNCPoint3[23805] = {X 196.8689, Y 47.1581, Z -4.6667, A 0.000, B 0.000, C 0.000 }
gfCNCPoint3[23806] = {X 195.0675, Y 47.9642, Z -4.6667, A 0.000, B 0.000, C 0.000 }
gfCNCPoint3[23807] = {X 193.2146, Y 48.6438, Z -4.6667, A 0.000, B 0.000, C 0.000 }
gfCNCPoint3[23808] = {X 191.3193, Y 49.1936, Z -4.6667, A 0.000, B 0.000, C 0.000 }
gfCNCPoint3[23809] = {X 189.3899, Y 49.5845, Z -4.6667, A 0.000, B 0.000, C 0.000 }
gfCNCPoint3[23810] = {X 187.4338, Y 49.8052, Z -4.6667, A 0.000, B 0.000, C 0.000 }
gfCNCPoint3[23811] = {X 185.4658, Y 49.8539, Z -4.6667, A 0.000, B 0.000, C 0.000 }
gfCNCPoint3[23812] = {X 183.5011, Y 49.7304, Z -4.6667, A 0.000, B 0.000, C 0.000 }
gfCNCPoint3[23813] = {X 181.5548, Y 49.4356, Z -4.6667, A 0.000, B 0.000, C 0.000 }
gfCNCPoint3[23814] = {X 179.6859, Y 48.9685, Z -4.6667, A 0.000, B 0.000, C 0.000 }
gfCNCPoint3[23815] = {X 177.8824, Y 48.2914, Z -4.6667, A 0.000, B 0.000, C 0.000 }
gfCNCPoint3[23816] = {X 176.1678, Y 47.4132, Z -4.6667, A 0.000, B 0.000, C 0.000 }
gfCNCPoint3[23817] = {X 174.5645, Y 46.3453, Z -4.6667, A 0.000, B 0.000, C 0.000 }
gfCNCPoint3[23818] = {X 173.3462, Y 45.3170, Z -4.6667, A 0.000, B 0.000, C 0.000 }
gfCNCPoint3[23819] = {X 172.2621, Y 44.1482, Z -4.6667, A 0.000, B 0.000, C 0.000 }
gfCNCPoint3[23820] = {X 171.3283, Y 42.8561, Z -4.6667, A 0.000, B 0.000, C 0.000 }
gfCNCPoint3[23821] = {X 170.5586, Y 41.4600, Z -4.6667, A 0.000, B 0.000, C 0.000 }
gfCNCPoint3[23822] = {X 169.9646, Y 39.9806, Z -4.6667, A 0.000, B 0.000, C 0.000 }
gfCNCPoint3[23823] = {X 169.5550, Y 38.4399, Z -4.6667, A 0.000, B 0.000, C 0.000 }
gfCNCPoint3[23824] = {X 169.3359, Y 36.8608, Z -4.6667, A 0.000, B 0.000, C 0.000 }
gfCNCPoint3[23825] = {X 169.2526, Y 35.0460, Z -4.6667, A 0.000, B 0.000, C 0.000 }
gfCNCPoint3[23826] = {X 169.3972, Y 33.2350, Z -4.6667, A 0.000, B 0.000, C 0.000 }
gfCNCPoint3[23827] = {X 169.7675, Y 31.4565, Z -4.6667, A 0.000, B 0.000, C 0.000 }
gfCNCPoint3[23828] = {X 170.3575, Y 29.7382, Z -4.6667, A 0.000, B 0.000, C 0.000 }
gfCNCPoint3[23829] = {X 171.0241, Y 28.3864, Z -4.6667, A 0.000, B 0.000, C 0.000 }
gfCNCPoint3[23830] = {X 171.8740, Y 27.1416, Z -4.6667, A 0.000, B 0.000, C 0.000 }
gfCNCPoint3[23831] = {X 172.8904, Y 26.0286, Z -4.6667, A 0.000, B 0.000, C 0.000 }
gfCNCPoint3[23832] = {X 174.0531, Y 25.0695, Z -4.6667, A 0.000, B 0.000, C 0.000 }
gfCNCPoint3[23833] = {X 175.3391, Y 24.2833, Z -4.6667, A 0.000, B 0.000, C 0.000 }
gfCNCPoint3[23834] = {X 174.4748, Y 23.9353, Z -4.6667, A 0.000, B 0.000, C 0.000 }
gfCNCPoint3[23835] = {X 173.7097, Y 23.4036, Z -4.6667, A 0.000, B 0.000, C 0.000 }
gfCNCPoint3[23836] = {X 173.0821, Y 22.7149, Z -4.6667, A 0.000, B 0.000, C 0.000 }
gfCNCPoint3[23837] = {X 172.6235, Y 21.9039, Z -4.6667, A 0.000, B 0.000, C 0.000 }
gfCNCPoint3[23838] = {X 171.3062, Y 18.6783, Z -4.6667, A 0.000, B 0.000, C 0.000 }
gfCNCPoint3[23839] = {X 167.6031, Y 20.1905, Z -4.6667, A 0.000, B 0.000, C 0.000 }
gfCNCPoint3[23840] = {X 171.3803, Y 18.6480, Z -4.6667, A 0.000, B 0.000, C 0.000 }
gfCNCPoint3[23841] = {X 170.0626, Y 15.4213, Z -4.6667, A 0.000, B 0.000, C 0.000 }
gfCNCPoint3[23842] = {X 169.8043, Y 14.4793, Z -4.6667, A 0.000, B 0.000, C 0.000 }
gfCNCPoint3[23843] = {X 169.7773, Y 13.5028, Z -4.6667, A 0.000, B 0.000, C 0.000 }
gfCNCPoint3[23844] = {X 169.9832, Y 12.5479, Z -4.6667, A 0.000, B 0.000, C 0.000 }
gfCNCPoint3[23845] = {X 170.4102, Y 11.6694, Z -4.6667, A 0.000, B 0.000, C 0.000 }
gfCNCPoint3[23846] = {X 171.0337, Y 10.9174, Z -4.6667, A 0.000, B 0.000, C 0.000 }
gfCNCPoint3[23847] = {X 171.8181, Y 10.3353, Z -4.6667, A 0.000, B 0.000, C 0.000 }
gfCNCPoint3[23848] = {X 172.4475, Y 9.9764, Z -4.6667, A 0.000, B 0.000, C 0.000 }
gfCNCPoint3[23849] = {X 173.3053, Y 9.6186, Z -4.6667, A 0.000, B 0.000, C 0.000 }
gfCNCPoint3[23850] = {X 174.2217, Y 9.4641, Z -4.6667, A 0.000, B 0.000, C 0.000 }
gfCNCPoint3[23851] = {X 175.1494, Y 9.5211, Z -4.6667, A 0.000, B 0.000, C 0.000 }
gfCNCPoint3[23852] = {X 176.0401, Y 9.7866, Z -4.6667, A 0.000, B 0.000, C 0.000 }
gfCNCPoint3[23853] = {X 177.9055, Y 8.9755, Z -4.6667, A 0.000, B 0.000, C 0.000 }
gfCNCPoint3[23854] = {X 179.8342, Y 8.3290, Z -4.6667, A 0.000, B 0.000, C 0.000 }
gfCNCPoint3[23855] = {X 181.8116, Y 7.8519, Z -4.6667, A 0.000, B 0.000, C 0.000 }
gfCNCPoint3[23856] = {X 183.8228, Y 7.5478, Z -4.6667, A 0.000, B 0.000, C 0.000 }
gfCNCPoint3[23857] = {X 185.8529, Y 7.4189, Z -4.6667, A 0.000, B 0.000, C 0.000 }
gfCNCPoint3[23858] = {X 187.8865, Y 7.4663, Z -4.6667, A 0.000, B 0.000, C 0.000 }
gfCNCPoint3[23859] = {X 189.9083, Y 7.6895, Z -4.6667, A 0.000, B 0.000, C 0.000 }
gfCNCPoint3[23860] = {X 191.6415, Y 8.0458, Z -4.6667, A 0.000, B 0.000, C 0.000 }
gfCNCPoint3[23861] = {X 193.3290, Y 8.5783, Z -4.6667, A 0.000, B 0.000, C 0.000 }
gfCNCPoint3[23862] = {X 194.9528, Y 9.2812, Z -4.6667, A 0.000, B 0.000, C 0.000 }
gfCNCPoint3[23863] = {X 196.4959, Y 10.1473, Z -4.6667, A 0.000, B 0.000, C 0.000 }
gfCNCPoint3[23864] = {X 197.9418, Y 11.1673, Z -4.6667, A 0.000, B 0.000, C 0.000 }
gfCNCPoint3[23865] = {X 199.2255, Y 12.3412, Z -4.6667, A 0.000, B 0.000, C 0.000 }
gfCNCPoint3[23866] = {X 200.3380, Y 13.6785, Z -4.6667, A 0.000, B 0.000, C 0.000 }
gfCNCPoint3[23867] = {X 201.2587, Y 15.1544, Z -4.6667, A 0.000, B 0.000, C 0.000 }
gfCNCPoint3[23868] = {X 201.9704, Y 16.7417, Z -4.6667, A 0.000, B 0.000, C 0.000 }
gfCNCPoint3[23869] = {X 202.4366, Y 18.3713, Z -4.6667, A 0.000, B 0.000, C 0.000 }
gfCNCPoint3[23870] = {X 202.7133, Y 20.0435, Z -4.6667, A 0.000, B 0.000, C 0.000 }
gfCNCPoint3[23871] = {X 202.7967, Y 21.7363, Z -4.6667, A 0.000, B 0.000, C 0.000 }
gfCNCPoint3[23872] = {X 202.6858, Y 23.4277, Z -4.6667, A 0.000, B 0.000, C 0.000 }
gfCNCPoint3[23873] = {X 202.3820, Y 25.0951, Z -4.6667, A 0.000, B 0.000, C 0.000 }
gfCNCPoint3[23874] = {X 201.9148, Y 26.6018, Z -4.6667, A 0.000, B 0.000, C 0.000 }
gfCNCPoint3[23875] = {X 201.2451, Y 28.0301, Z -4.6667, A 0.000, B 0.000, C 0.000 }
gfCNCPoint3[23876] = {X 200.3854, Y 29.3527, Z -4.6667, A 0.000, B 0.000, C 0.000 }
gfCNCPoint3[23877] = {X 199.3521, Y 30.5447, Z -4.6667, A 0.000, B 0.000, C 0.000 }
gfCNCPoint3[23878] = {X 198.1649, Y 31.5834, Z -4.6667, A 0.000, B 0.000, C 0.000 }
gfCNCPoint3[23879] = {X 199.0629, Y 31.8621, Z -4.6667, A 0.000, B 0.000, C 0.000 }
gfCNCPoint3[23880] = {X 199.8732, Y 32.3389, Z -4.6667, A 0.000, B 0.000, C 0.000 }
gfCNCPoint3[23881] = {X 200.5528, Y 32.9886, Z -4.6667, A 0.000, B 0.000, C 0.000 }
gfCNCPoint3[23882] = {X 201.0657, Y 33.7766, Z -4.6667, A 0.000, B 0.000, C 0.000 }
gfCNCPoint3[23883] = {X 204.1061, Y 40.0576, Z -4.6667, A 0.000, B 0.000, C 0.000 }
gfCNCPoint3[23884] = {X 204.4089, Y 40.9162, Z -4.6667, A 0.000, B 0.000, C 0.000 }
gfCNCPoint3[23885] = {X 204.5137, Y 41.8206, Z -4.6667, A 0.000, B 0.000, C 0.000 }
gfCNCPoint3[23886] = {X 204.4154, Y 42.7257, Z -4.6667, A 0.000, B 0.000, C 0.000 }
gfCNCPoint3[23887] = {X 204.1188, Y 43.5864, Z -4.6667, A 0.000, B 0.000, C 0.000 }
gfCNCPoint3[23888] = {X 203.6387, Y 44.3600, Z -4.6667, A 0.000, B 0.000, C 0.000 }
gfCNCPoint3[23889] = {X 202.9990, Y 45.0078, Z -4.6667, A 0.000, B 0.000, C 0.000 }
gfCNCPoint3[23890] = {X 202.4628, Y 45.4413, Z -4.6667, A 0.000, B 0.000, C 0.000 }
gfCNCPoint3[23891] = {X 201.7790, Y 45.8890, Z -4.6667, A 0.000, B 0.000, C 0.000 }
gfCNCPoint3[23892] = {X 201.0199, Y 46.1919, Z -4.6667, A 0.000, B 0.000, C 0.000 }
gfCNCPoint3[23893] = {X 200.2158, Y 46.3378, Z -4.6667, A 0.000, B 0.000, C 0.000 }
gfCNCPoint3[23894] = {X 199.3987, Y 46.3211, Z -4.6667, A 0.000, B 0.000, C 0.000 }
gfCNCPoint3[23895] = {X 198.6012, Y 46.1423, Z -4.6667, A 0.000, B 0.000, C 0.000 }
gfCNCPoint3[23896] = {X 196.8578, Y 47.0745, Z -4.6667, A 0.000, B 0.000, C 0.000 }
gfCNCPoint3[23897] = {X 195.0539, Y 47.8833, Z -4.6667, A 0.000, B 0.000, C 0.000 }
gfCNCPoint3[23898] = {X 193.1982, Y 48.5650, Z -4.6667, A 0.000, B 0.000, C 0.000 }
gfCNCPoint3[23899] = {X 191.2996, Y 49.1161, Z -4.6667, A 0.000, B 0.000, C 0.000 }
gfCNCPoint3[23900] = {X 189.3772, Y 49.5055, Z -4.6667, A 0.000, B 0.000, C 0.000 }
gfCNCPoint3[23901] = {X 187.4280, Y 49.7254, Z -4.6667, A 0.000, B 0.000, C 0.000 }
gfCNCPoint3[23902] = {X 185.4671, Y 49.7740, Z -4.6667, A 0.000, B 0.000, C 0.000 }
gfCNCPoint3[23903] = {X 183.5094, Y 49.6509, Z -4.6667, A 0.000, B 0.000, C 0.000 }
gfCNCPoint3[23904] = {X 181.5700, Y 49.3571, Z -4.6667, A 0.000, B 0.000, C 0.000 }
gfCNCPoint3[23905] = {X 179.7098, Y 48.8921, Z -4.6667, A 0.000, B 0.000, C 0.000 }
gfCNCPoint3[23906] = {X 177.9148, Y 48.2182, Z -4.6667, A 0.000, B 0.000, C 0.000 }
gfCNCPoint3[23907] = {X 176.2082, Y 47.3441, Z -4.6667, A 0.000, B 0.000, C 0.000 }
gfCNCPoint3[23908] = {X 174.6124, Y 46.2812, Z -4.6667, A 0.000, B 0.000, C 0.000 }
gfCNCPoint3[23909] = {X 173.4014, Y 45.2591, Z -4.6667, A 0.000, B 0.000, C 0.000 }
gfCNCPoint3[23910] = {X 172.3238, Y 44.0973, Z -4.6667, A 0.000, B 0.000, C 0.000 }
gfCNCPoint3[23911] = {X 171.3956, Y 42.8129, Z -4.6667, A 0.000, B 0.000, C 0.000 }
gfCNCPoint3[23912] = {X 170.6306, Y 41.4251, Z -4.6667, A 0.000, B 0.000, C 0.000 }
gfCNCPoint3[23913] = {X 170.0402, Y 39.9545, Z -4.6667, A 0.000, B 0.000, C 0.000 }
gfCNCPoint3[23914] = {X 169.6332, Y 38.4230, Z -4.6667, A 0.000, B 0.000, C 0.000 }
gfCNCPoint3[23915] = {X 169.4156, Y 36.8534, Z -4.6667, A 0.000, B 0.000, C 0.000 }
gfCNCPoint3[23916] = {X 169.3326, Y 35.0482, Z -4.6667, A 0.000, B 0.000, C 0.000 }
gfCNCPoint3[23917] = {X 169.4764, Y 33.2469, Z -4.6667, A 0.000, B 0.000, C 0.000 }
gfCNCPoint3[23918] = {X 169.8446, Y 31.4778, Z -4.6667, A 0.000, B 0.000, C 0.000 }
gfCNCPoint3[23919] = {X 170.4315, Y 29.7687, Z -4.6667, A 0.000, B 0.000, C 0.000 }
gfCNCPoint3[23920] = {X 171.1147, Y 28.3899, Z -4.6667, A 0.000, B 0.000, C 0.000 }
gfCNCPoint3[23921] = {X 171.9900, Y 27.1244, Z -4.6667, A 0.000, B 0.000, C 0.000 }
gfCNCPoint3[23922] = {X 173.0390, Y 25.9987, Z -4.6667, A 0.000, B 0.000, C 0.000 }
gfCNCPoint3[23923] = {X 174.2397, Y 25.0364, Z -4.6667, A 0.000, B 0.000, C 0.000 }
gfCNCPoint3[23924] = {X 175.5669, Y 24.2577, Z -4.6667, A 0.000, B 0.000, C 0.000 }
gfCNCPoint3[23925] = {X 174.6548, Y 23.9380, Z -4.6667, A 0.000, B 0.000, C 0.000 }
gfCNCPoint3[23926] = {X 173.8436, Y 23.4127, Z -4.6667, A 0.000, B 0.000, C 0.000 }
gfCNCPoint3[23927] = {X 173.1786, Y 22.7112, Z -4.6667, A 0.000, B 0.000, C 0.000 }
gfCNCPoint3[23928] = {X 172.6973, Y 21.8731, Z -4.6667, A 0.000, B 0.000, C 0.000 }
gfCNCPoint3[23929] = {X 171.3803, Y 18.6480, Z -4.6667, A 0.000, B 0.000, C 0.000 }
gfCNCPoint3[23930] = {X 167.6770, Y 20.1603, Z -4.6667, A 0.000, B 0.000, C 0.000 }
gfCNCPoint3[23931] = {X 167.6769, Y 20.1601, Z -4.6667, A 0.000, B 0.000, C 0.000 }
gfCNCPoint3[23932] = {X 171.4542, Y 18.6179, Z -4.6667, A 0.000, B 0.000, C 0.000 }
gfCNCPoint3[23933] = {X 170.1367, Y 15.3911, Z -4.6667, A 0.000, B 0.000, C 0.000 }
gfCNCPoint3[23934] = {X 169.8835, Y 14.4675, Z -4.6667, A 0.000, B 0.000, C 0.000 }
gfCNCPoint3[23935] = {X 169.8570, Y 13.5102, Z -4.6667, A 0.000, B 0.000, C 0.000 }
gfCNCPoint3[23936] = {X 170.0588, Y 12.5740, Z -4.6667, A 0.000, B 0.000, C 0.000 }
gfCNCPoint3[23937] = {X 170.4774, Y 11.7127, Z -4.6667, A 0.000, B 0.000, C 0.000 }
gfCNCPoint3[23938] = {X 171.0888, Y 10.9755, Z -4.6667, A 0.000, B 0.000, C 0.000 }
gfCNCPoint3[23939] = {X 171.8578, Y 10.4048, Z -4.6667, A 0.000, B 0.000, C 0.000 }
gfCNCPoint3[23940] = {X 172.4867, Y 10.0462, Z -4.6667, A 0.000, B 0.000, C 0.000 }
gfCNCPoint3[23941] = {X 173.3363, Y 9.6929, Z -4.6667, A 0.000, B 0.000, C 0.000 }
gfCNCPoint3[23942] = {X 174.2443, Y 9.5431, Z -4.6667, A 0.000, B 0.000, C 0.000 }
gfCNCPoint3[23943] = {X 175.1624, Y 9.6048, Z -4.6667, A 0.000, B 0.000, C 0.000 }
gfCNCPoint3[23944] = {X 176.0421, Y 9.8746, Z -4.6667, A 0.000, B 0.000, C 0.000 }
gfCNCPoint3[23945] = {X 177.9048, Y 9.0615, Z -4.6667, A 0.000, B 0.000, C 0.000 }
gfCNCPoint3[23946] = {X 179.8311, Y 8.4132, Z -4.6667, A 0.000, B 0.000, C 0.000 }
gfCNCPoint3[23947] = {X 181.8063, Y 7.9345, Z -4.6667, A 0.000, B 0.000, C 0.000 }
gfCNCPoint3[23948] = {X 183.8157, Y 7.6290, Z -4.6667, A 0.000, B 0.000, C 0.000 }
gfCNCPoint3[23949] = {X 185.8440, Y 7.4991, Z -4.6667, A 0.000, B 0.000, C 0.000 }
gfCNCPoint3[23950] = {X 187.8759, Y 7.5458, Z -4.6667, A 0.000, B 0.000, C 0.000 }
gfCNCPoint3[23951] = {X 189.8961, Y 7.7686, Z -4.6667, A 0.000, B 0.000, C 0.000 }
gfCNCPoint3[23952] = {X 191.6213, Y 8.1232, Z -4.6667, A 0.000, B 0.000, C 0.000 }
gfCNCPoint3[23953] = {X 193.3009, Y 8.6532, Z -4.6667, A 0.000, B 0.000, C 0.000 }
gfCNCPoint3[23954] = {X 194.9173, Y 9.3529, Z -4.6667, A 0.000, B 0.000, C 0.000 }
gfCNCPoint3[23955] = {X 196.4531, Y 10.2149, Z -4.6667, A 0.000, B 0.000, C 0.000 }
gfCNCPoint3[23956] = {X 197.8924, Y 11.2302, Z -4.6667, A 0.000, B 0.000, C 0.000 }
gfCNCPoint3[23957] = {X 199.1678, Y 12.3966, Z -4.6667, A 0.000, B 0.000, C 0.000 }
gfCNCPoint3[23958] = {X 200.2731, Y 13.7253, Z -4.6667, A 0.000, B 0.000, C 0.000 }
gfCNCPoint3[23959] = {X 201.1879, Y 15.1917, Z -4.6667, A 0.000, B 0.000, C 0.000 }
gfCNCPoint3[23960] = {X 201.8951, Y 16.7687, Z -4.6667, A 0.000, B 0.000, C 0.000 }
gfCNCPoint3[23961] = {X 202.3587, Y 18.3894, Z -4.6667, A 0.000, B 0.000, C 0.000 }
gfCNCPoint3[23962] = {X 202.6338, Y 20.0525, Z -4.6667, A 0.000, B 0.000, C 0.000 }
gfCNCPoint3[23963] = {X 202.7167, Y 21.7361, Z -4.6667, A 0.000, B 0.000, C 0.000 }
gfCNCPoint3[23964] = {X 202.6064, Y 23.4182, Z -4.6667, A 0.000, B 0.000, C 0.000 }
gfCNCPoint3[23965] = {X 202.3042, Y 25.0766, Z -4.6667, A 0.000, B 0.000, C 0.000 }
gfCNCPoint3[23966] = {X 201.8267, Y 26.6077, Z -4.6667, A 0.000, B 0.000, C 0.000 }
gfCNCPoint3[23967] = {X 201.1385, Y 28.0565, Z -4.6667, A 0.000, B 0.000, C 0.000 }
gfCNCPoint3[23968] = {X 200.2534, Y 29.3941, Z -4.6667, A 0.000, B 0.000, C 0.000 }
gfCNCPoint3[23969] = {X 199.1889, Y 30.5938, Z -4.6667, A 0.000, B 0.000, C 0.000 }
gfCNCPoint3[23970] = {X 197.9663, Y 31.6319, Z -4.6667, A 0.000, B 0.000, C 0.000 }
gfCNCPoint3[23971] = {X 198.7280, Y 31.8159, Z -4.6667, A 0.000, B 0.000, C 0.000 }
gfCNCPoint3[23972] = {X 199.4393, Y 32.1449, Z -4.6667, A 0.000, B 0.000, C 0.000 }
gfCNCPoint3[23973] = {X 200.0727, Y 32.6062, Z -4.6667, A 0.000, B 0.000, C 0.000 }
gfCNCPoint3[23974] = {X 200.6041, Y 33.1822, Z -4.6667, A 0.000, B 0.000, C 0.000 }
gfCNCPoint3[23975] = {X 201.0129, Y 33.8507, Z -4.6667, A 0.000, B 0.000, C 0.000 }
gfCNCPoint3[23976] = {X 204.0341, Y 40.0925, Z -4.6667, A 0.000, B 0.000, C 0.000 }
gfCNCPoint3[23977] = {X 204.3309, Y 40.9342, Z -4.6667, A 0.000, B 0.000, C 0.000 }
gfCNCPoint3[23978] = {X 204.4337, Y 41.8209, Z -4.6667, A 0.000, B 0.000, C 0.000 }
gfCNCPoint3[23979] = {X 204.3373, Y 42.7082, Z -4.6667, A 0.000, B 0.000, C 0.000 }
gfCNCPoint3[23980] = {X 204.0465, Y 43.5521, Z -4.6667, A 0.000, B 0.000, C 0.000 }
gfCNCPoint3[23981] = {X 203.5758, Y 44.3105, Z -4.6667, A 0.000, B 0.000, C 0.000 }
gfCNCPoint3[23982] = {X 202.9487, Y 44.9456, Z -4.6667, A 0.000, B 0.000, C 0.000 }
gfCNCPoint3[23983] = {X 202.4125, Y 45.3791, Z -4.6667, A 0.000, B 0.000, C 0.000 }
gfCNCPoint3[23984] = {X 201.7357, Y 45.8213, Z -4.6667, A 0.000, B 0.000, C 0.000 }
gfCNCPoint3[23985] = {X 200.9840, Y 46.1189, Z -4.6667, A 0.000, B 0.000, C 0.000 }
gfCNCPoint3[23986] = {X 200.1879, Y 46.2597, Z -4.6667, A 0.000, B 0.000, C 0.000 }
gfCNCPoint3[23987] = {X 199.3798, Y 46.2381, Z -4.6667, A 0.000, B 0.000, C 0.000 }
gfCNCPoint3[23988] = {X 198.5923, Y 46.0549, Z -4.6667, A 0.000, B 0.000, C 0.000 }
gfCNCPoint3[23989] = {X 196.8469, Y 46.9907, Z -4.6667, A 0.000, B 0.000, C 0.000 }
gfCNCPoint3[23990] = {X 195.0405, Y 47.8024, Z -4.6667, A 0.000, B 0.000, C 0.000 }
gfCNCPoint3[23991] = {X 193.1818, Y 48.4861, Z -4.6667, A 0.000, B 0.000, C 0.000 }
gfCNCPoint3[23992] = {X 191.2800, Y 49.0385, Z -4.6667, A 0.000, B 0.000, C 0.000 }
gfCNCPoint3[23993] = {X 189.3644, Y 49.4265, Z -4.6667, A 0.000, B 0.000, C 0.000 }
gfCNCPoint3[23994] = {X 187.4222, Y 49.6456, Z -4.6667, A 0.000, B 0.000, C 0.000 }
gfCNCPoint3[23995] = {X 185.4683, Y 49.6940, Z -4.6667, A 0.000, B 0.000, C 0.000 }
gfCNCPoint3[23996] = {X 183.5177, Y 49.5713, Z -4.6667, A 0.000, B 0.000, C 0.000 }
gfCNCPoint3[23997] = {X 181.5852, Y 49.2785, Z -4.6667, A 0.000, B 0.000, C 0.000 }
gfCNCPoint3[23998] = {X 179.7338, Y 48.8158, Z -4.6667, A 0.000, B 0.000, C 0.000 }
gfCNCPoint3[23999] = {X 177.9472, Y 48.1451, Z -4.6667, A 0.000, B 0.000, C 0.000 }
gfCNCPoint3[24000] = {X 176.2487, Y 47.2751, Z -4.6667, A 0.000, B 0.000, C 0.000 }
gfCNCPoint3[24001] = {X 174.6604, Y 46.2172, Z -4.6667, A 0.000, B 0.000, C 0.000 }
gfCNCPoint3[24002] = {X 173.4567, Y 45.2013, Z -4.6667, A 0.000, B 0.000, C 0.000 }
gfCNCPoint3[24003] = {X 172.3855, Y 44.0464, Z -4.6667, A 0.000, B 0.000, C 0.000 }
gfCNCPoint3[24004] = {X 171.4629, Y 42.7698, Z -4.6667, A 0.000, B 0.000, C 0.000 }
gfCNCPoint3[24005] = {X 170.7026, Y 41.3903, Z -4.6667, A 0.000, B 0.000, C 0.000 }
gfCNCPoint3[24006] = {X 170.1159, Y 39.9285, Z -4.6667, A 0.000, B 0.000, C 0.000 }
gfCNCPoint3[24007] = {X 169.7114, Y 38.4062, Z -4.6667, A 0.000, B 0.000, C 0.000 }
gfCNCPoint3[24008] = {X 169.4953, Y 36.8460, Z -4.6667, A 0.000, B 0.000, C 0.000 }
